LIN {X 0,Y 531.039,Z 315.337,A -85,B 0,C 180,E1 -4242.225,E2 -4242.225} C_VEL
LIN {X 0,Y 530.994,Z 315.34,A -85,B 0,C 180,E1 -4245.35,E2 -4245.35} C_VEL
LIN {X 0,Y 530.991,Z 315.339,A -85,B 0,C 180,E1 -4248.521,E2 -4248.521} C_VEL
LIN {X 0,Y 530.998,Z 315.337,A -85,B 0,C 180,E1 -4250.938,E2 -4250.938} C_VEL
LIN {X 0,Y 530.979,Z 315.343,A -85,B 0,C 180,E1 -4254.225,E2 -4254.225} C_VEL
LIN {X 0,Y 531.004,Z 315.337,A -85,B 0,C 180,E1 -4256.744,E2 -4256.744} C_VEL
LIN {X 0,Y 530.981,Z 315.343,A -85,B 0,C 180,E1 -4259.323,E2 -4259.323} C_VEL
LIN {X 0,Y 530.97,Z 315.344,A -85,B 0,C 180,E1 -4262.102,E2 -4262.102} C_VEL
LIN {X 0,Y 530.986,Z 315.339,A -85,B 0,C 180,E1 -4264.854,E2 -4264.854} C_VEL
LIN {X 0,Y 530.966,Z 315.347,A -85,B 0,C 180,E1 -4267.508,E2 -4267.508} C_VEL
LIN {X 0,Y 530.982,Z 315.34,A -85,B 0,C 180,E1 -4270.433,E2 -4270.433} C_VEL
LIN {X 0,Y 530.961,Z 315.347,A -85,B 0,C 180,E1 -4273.282,E2 -4273.282} C_VEL
LIN {X 0,Y 530.982,Z 315.347,A -85,B 0,C 180,E1 -4275.622,E2 -4275.622} C_VEL
LIN {X 0,Y 530.994,Z 315.338,A -85,B 0,C 180,E1 -4278.565,E2 -4278.565} C_VEL
LIN {X 0,Y 530.958,Z 315.35,A -85,B 0,C 180,E1 -4281.53,E2 -4281.53} C_VEL
LIN {X 0,Y 530.955,Z 315.343,A -85,B 0,C 180,E1 -4284.381,E2 -4284.381} C_VEL
LIN {X 0,Y 530.968,Z 315.345,A -85,B 0,C 180,E1 -4287.134,E2 -4287.134} C_VEL
LIN {X 0,Y 530.964,Z 315.346,A -85,B 0,C 180,E1 -4289.803,E2 -4289.803} C_VEL
LIN {X 0,Y 531.013,Z 315.335,A -85,B 0,C 180,E1 -4292.469,E2 -4292.469} C_VEL
LIN {X 0,Y 531.002,Z 315.339,A -85,B 0,C 180,E1 -4294.943,E2 -4294.943} C_VEL
LIN {X 0,Y 530.969,Z 315.349,A -85,B 0,C 180,E1 -4297.377,E2 -4297.377} C_VEL
LIN {X 0,Y 532.621,Z 320.667,A -85,B 0,C 180,E1 -4297.507,E2 -4297.507} C_VEL
LIN {X 0,Y 532.362,Z 402.902,A -85,B 0,C 180,E1 -4298.663,E2 -4298.663} C_VEL
LIN {X 0,Y 532.209,Z 415.998,A -85,B 0,C 180,E1 -4298.986,E2 -4298.986} C_VEL
LIN {X 0,Y 532.03,Z 429.878,A -85,B 0,C 180,E1 -4299.517,E2 -4299.517} C_VEL
LIN {X 0,Y 531.847,Z 441.157,A -85,B 0,C 180,E1 -4300.107,E2 -4300.107} C_VEL
LIN {X 0,Y 531.61,Z 451.611,A -85,B 0,C 180,E1 -4300.801,E2 -4300.801} C_VEL
LIN {X 0,Y 531.404,Z 461.288,A -85,B 0,C 180,E1 -4301.594,E2 -4301.594} C_VEL
LIN {X 0,Y 531.176,Z 470.826,A -85,B 0,C 180,E1 -4302.552,E2 -4302.552} C_VEL
LIN {X 0,Y 530.961,Z 479.751,A -85,B 0,C 180,E1 -4303.664,E2 -4303.664} C_VEL
LIN {X 0,Y 530.809,Z 487.195,A -85,B 0,C 180,E1 -4304.83,E2 -4304.83} C_VEL
LIN {X 0,Y 530.705,Z 492.339,A -85,B 0,C 180,E1 -4305.819,E2 -4305.819} C_VEL
LIN {X 0,Y 530.574,Z 497.221,A -85,B 0,C 180,E1 -4306.987,E2 -4306.987} C_VEL
LIN {X 0,Y 530.558,Z 500.943,A -85,B 0,C 180,E1 -4308.152,E2 -4308.152} C_VEL
LIN {X 0,Y 530.478,Z 503.626,A -85,B 0,C 180,E1 -4309.311,E2 -4309.311} C_VEL
LIN {X 0,Y 530.462,Z 504.893,A -85,B 0,C 180,E1 -4310.083,E2 -4310.083} C_VEL
LIN {X 0,Y 530.464,Z 505.756,A -85,B 0,C 180,E1 -4310.852,E2 -4310.852} C_VEL
LIN {X 0,Y 530.493,Z 506.174,A -85,B 0,C 180,E1 -4312.387,E2 -4312.387} C_VEL
LIN {X 0,Y 530.548,Z 505.548,A -85,B 0,C 180,E1 -4313.468,E2 -4313.468} C_VEL
LIN {X 0,Y 530.506,Z 503.888,A -85,B 0,C 180,E1 -4314.679,E2 -4314.679} C_VEL
LIN {X 0,Y 530.559,Z 501.365,A -85,B 0,C 180,E1 -4315.822,E2 -4315.822} C_VEL
LIN {X 0,Y 530.61,Z 497.858,A -85,B 0,C 180,E1 -4316.963,E2 -4316.963} C_VEL
LIN {X 0,Y 530.664,Z 493.275,A -85,B 0,C 180,E1 -4318.103,E2 -4318.103} C_VEL
LIN {X 0,Y 530.832,Z 487.475,A -85,B 0,C 180,E1 -4319.242,E2 -4319.242} C_VEL
LIN {X 0,Y 530.951,Z 480.294,A -85,B 0,C 180,E1 -4320.38,E2 -4320.38} C_VEL
LIN {X 0,Y 531.189,Z 471.278,A -85,B 0,C 180,E1 -4321.517,E2 -4321.517} C_VEL
LIN {X 0,Y 531.409,Z 461.946,A -85,B 0,C 180,E1 -4322.464,E2 -4322.464} C_VEL
LIN {X 0,Y 531.655,Z 452.816,A -85,B 0,C 180,E1 -4323.221,E2 -4323.221} C_VEL
LIN {X 0,Y 531.875,Z 443.079,A -85,B 0,C 180,E1 -4323.883,E2 -4323.883} C_VEL
LIN {X 0,Y 532.06,Z 431.73,A -85,B 0,C 180,E1 -4324.499,E2 -4324.499} C_VEL
LIN {X 0,Y 532.19,Z 418.807,A -85,B 0,C 180,E1 -4325.019,E2 -4325.019} C_VEL
LIN {X 0,Y 532.304,Z 405.636,A -85,B 0,C 180,E1 -4325.374,E2 -4325.374} C_VEL
LIN {X 0,Y 532.466,Z 376.911,A -85,B 0,C 180,E1 -4325.8,E2 -4325.8} C_VEL
LIN {X 0,Y 532.689,Z 320.761,A -85,B 0,C 180,E1 -4326.582,E2 -4326.582} C_VEL
LIN {X 0,Y 531.014,Z 315.344,A -85,B 0,C 180,E1 -4326.714,E2 -4326.714} C_VEL
LIN {X 0,Y 530.993,Z 315.343,A -85,B 0,C 180,E1 -4329.139,E2 -4329.139} C_VEL
LIN {X 0,Y 530.972,Z 315.347,A -85,B 0,C 180,E1 -4332.227,E2 -4332.227} C_VEL
LIN {X 0,Y 530.987,Z 315.34,A -85,B 0,C 180,E1 -4335.35,E2 -4335.35} C_VEL
LIN {X 0,Y 530.95,Z 315.351,A -85,B 0,C 180,E1 -4338.523,E2 -4338.523} C_VEL
LIN {X 0,Y 530.931,Z 315.349,A -85,B 0,C 180,E1 -4340.941,E2 -4340.941} C_VEL
LIN {X 0,Y 530.947,Z 315.344,A -85,B 0,C 180,E1 -4343.397,E2 -4343.397} C_VEL
LIN {X 0,Y 530.93,Z 315.351,A -85,B 0,C 180,E1 -4345.902,E2 -4345.902} C_VEL
LIN {X 0,Y 530.933,Z 315.351,A -85,B 0,C 180,E1 -4348.46,E2 -4348.46} C_VEL
LIN {X 0,Y 530.944,Z 315.344,A -85,B 0,C 180,E1 -4351.08,E2 -4351.08} C_VEL
LIN {X 0,Y 530.955,Z 315.347,A -85,B 0,C 180,E1 -4353.775,E2 -4353.775} C_VEL
LIN {X 0,Y 530.911,Z 315.349,A -85,B 0,C 180,E1 -4356.562,E2 -4356.562} C_VEL
LIN {X 0,Y 530.972,Z 315.342,A -85,B 0,C 180,E1 -4359.445,E2 -4359.445} C_VEL
LIN {X 0,Y 530.922,Z 315.348,A -85,B 0,C 180,E1 -4362.463,E2 -4362.463} C_VEL
LIN {X 0,Y 530.97,Z 315.344,A -85,B 0,C 180,E1 -4365.451,E2 -4365.451} C_VEL
LIN {X 0,Y 530.967,Z 315.341,A -85,B 0,C 180,E1 -4368.561,E2 -4368.561} C_VEL
LIN {X 0,Y 530.956,Z 315.349,A -85,B 0,C 180,E1 -4371.529,E2 -4371.529} C_VEL
LIN {X 0,Y 530.952,Z 315.344,A -85,B 0,C 180,E1 -4374.379,E2 -4374.379} C_VEL
LIN {X 0,Y 530.971,Z 315.344,A -85,B 0,C 180,E1 -4377.133,E2 -4377.133} C_VEL
LIN {X 0,Y 530.973,Z 315.347,A -85,B 0,C 180,E1 -4379.803,E2 -4379.803} C_VEL
LIN {X 0,Y 531.024,Z 315.545,A -85,B 0,C 180,E1 -4382.212,E2 -4382.212} C_VEL
LIN {X 0,Y 533.268,Z 326.124,A -85,B 0,C 180,E1 -4383.661,E2 -4383.661} C_VEL
LIN {X 0,Y 532.877,Z 345.545,A -85,B 0,C 180,E1 -4386.074,E2 -4386.074} C_VEL
LIN {X 0,Y 532.428,Z 368.596,A -85,B 0,C 180,E1 -4388.918,E2 -4388.918} C_VEL
LIN {X 0,Y 531.903,Z 396.768,A -85,B 0,C 180,E1 -4392.308,E2 -4392.308} C_VEL
LIN {X 0,Y 531.523,Z 420.074,A -85,B 0,C 180,E1 -4395.053,E2 -4395.053} C_VEL
LIN {X 0,Y 532.776,Z 431.286,A -85,B 0,C 180,E1 -4395.246,E2 -4395.246} C_VEL
LIN {X 0,Y 532.352,Z 528.112,A -85,B 0,C 180,E1 -4396.569,E2 -4396.569} C_VEL
LIN {X 0,Y 532.201,Z 540.608,A -85,B 0,C 180,E1 -4396.857,E2 -4396.857} C_VEL
LIN {X 0,Y 531.959,Z 553.505,A -85,B 0,C 180,E1 -4397.312,E2 -4397.312} C_VEL
LIN {X 0,Y 531.724,Z 565.811,A -85,B 0,C 180,E1 -4397.905,E2 -4397.905} C_VEL
LIN {X 0,Y 531.503,Z 577.756,A -85,B 0,C 180,E1 -4398.656,E2 -4398.656} C_VEL
LIN {X 0,Y 531.256,Z 588.623,A -85,B 0,C 180,E1 -4399.519,E2 -4399.519} C_VEL
LIN {X 0,Y 531.033,Z 598.418,A -85,B 0,C 180,E1 -4400.477,E2 -4400.477} C_VEL
LIN {X 0,Y 530.851,Z 606.454,A -85,B 0,C 180,E1 -4401.434,E2 -4401.434} C_VEL
LIN {X 0,Y 530.682,Z 614.305,A -85,B 0,C 180,E1 -4402.581,E2 -4402.581} C_VEL
LIN {X 0,Y 530.585,Z 621.541,A -85,B 0,C 180,E1 -4403.917,E2 -4403.917} C_VEL
LIN {X 0,Y 530.459,Z 626.318,A -85,B 0,C 180,E1 -4405.06,E2 -4405.06} C_VEL
LIN {X 0,Y 530.516,Z 629.946,A -85,B 0,C 180,E1 -4406.202,E2 -4406.202} C_VEL
LIN {X 0,Y 530.457,Z 631.803,A -85,B 0,C 180,E1 -4406.962,E2 -4406.962} C_VEL
LIN {X 0,Y 530.411,Z 633.192,A -85,B 0,C 180,E1 -4407.722,E2 -4407.722} C_VEL
LIN {X 0,Y 530.344,Z 634.785,A -85,B 0,C 180,E1 -4409.241,E2 -4409.241} C_VEL
LIN {X 0,Y 530.342,Z 635,A -85,B 0,C 180,E1 -4410,E2 -4410} C_VEL
LIN {X 0,Y 530.361,Z 634.183,A -85,B 0,C 180,E1 -4411.519,E2 -4411.519} C_VEL
LIN {X 0,Y 530.411,Z 633.195,A -85,B 0,C 180,E1 -4412.278,E2 -4412.278} C_VEL
LIN {X 0,Y 530.457,Z 631.807,A -85,B 0,C 180,E1 -4413.038,E2 -4413.038} C_VEL
LIN {X 0,Y 530.522,Z 628.876,A -85,B 0,C 180,E1 -4414.178,E2 -4414.178} C_VEL
LIN {X 0,Y 530.525,Z 624.876,A -85,B 0,C 180,E1 -4415.321,E2 -4415.321} C_VEL
LIN {X 0,Y 530.596,Z 619.076,A -85,B 0,C 180,E1 -4416.579,E2 -4416.579} C_VEL
LIN {X 0,Y 530.728,Z 611.833,A -85,B 0,C 180,E1 -4417.801,E2 -4417.801} C_VEL
LIN {X 0,Y 530.908,Z 603.357,A -85,B 0,C 180,E1 -4418.948,E2 -4418.948} C_VEL
LIN {X 0,Y 531.103,Z 594.649,A -85,B 0,C 180,E1 -4419.906,E2 -4419.906} C_VEL
LIN {X 0,Y 531.345,Z 583.897,A -85,B 0,C 180,E1 -4420.864,E2 -4420.864} C_VEL
LIN {X 0,Y 531.559,Z 572.848,A -85,B 0,C 180,E1 -4421.659,E2 -4421.659} C_VEL
LIN {X 0,Y 531.831,Z 561.541,A -85,B 0,C 180,E1 -4422.303,E2 -4422.303} C_VEL
LIN {X 0,Y 532.054,Z 549.413,A -85,B 0,C 180,E1 -4422.831,E2 -4422.831} C_VEL
LIN {X 0,Y 532.213,Z 536.317,A -85,B 0,C 180,E1 -4423.24,E2 -4423.24} C_VEL
LIN {X 0,Y 532.363,Z 524.159,A -85,B 0,C 180,E1 -4423.479,E2 -4423.479} C_VEL
LIN {X 0,Y 532.625,Z 428.755,A -85,B 0,C 180,E1 -4424.776,E2 -4424.776} C_VEL
LIN {X 0,Y 531.483,Z 418.906,A -85,B 0,C 180,E1 -4424.969,E2 -4424.969} C_VEL
LIN {X 0,Y 531.936,Z 388.838,A -85,B 0,C 180,E1 -4428.487,E2 -4428.487} C_VEL
LIN {X 0,Y 532.271,Z 363.451,A -85,B 0,C 180,E1 -4431.494,E2 -4431.494} C_VEL
LIN {X 0,Y 532.637,Z 339.943,A -85,B 0,C 180,E1 -4434.325,E2 -4434.325} C_VEL
LIN {X 0,Y 532.749,Z 324.506,A -85,B 0,C 180,E1 -4436.226,E2 -4436.226} C_VEL
LIN {X 0,Y 530.968,Z 315.346,A -85,B 0,C 180,E1 -4437.466,E2 -4437.466} C_VEL
LIN {X 0,Y 530.972,Z 315.349,A -85,B 0,C 180,E1 -4440.197,E2 -4440.197} C_VEL
LIN {X 0,Y 530.969,Z 315.346,A -85,B 0,C 180,E1 -4442.867,E2 -4442.867} C_VEL
LIN {X 0,Y 530.953,Z 315.345,A -85,B 0,C 180,E1 -4445.62,E2 -4445.62} C_VEL
LIN {X 0,Y 530.966,Z 315.347,A -85,B 0,C 180,E1 -4448.653,E2 -4448.653} C_VEL
LIN {X 0,Y 530.966,Z 315.343,A -85,B 0,C 180,E1 -4451.438,E2 -4451.438} C_VEL
LIN {X 0,Y 530.968,Z 315.345,A -85,B 0,C 180,E1 -4454.549,E2 -4454.549} C_VEL
LIN {X 0,Y 530.932,Z 315.348,A -85,B 0,C 180,E1 -4457.538,E2 -4457.538} C_VEL
LIN {X 0,Y 530.97,Z 315.343,A -85,B 0,C 180,E1 -4460.555,E2 -4460.555} C_VEL
LIN {X 0,Y 530.909,Z 315.35,A -85,B 0,C 180,E1 -4463.437,E2 -4463.437} C_VEL
LIN {X 0,Y 530.953,Z 315.347,A -85,B 0,C 180,E1 -4466.224,E2 -4466.224} C_VEL
LIN {X 0,Y 530.942,Z 315.345,A -85,B 0,C 180,E1 -4468.919,E2 -4468.919} C_VEL
LIN {X 0,Y 530.931,Z 315.352,A -85,B 0,C 180,E1 -4471.54,E2 -4471.54} C_VEL
LIN {X 0,Y 530.93,Z 315.35,A -85,B 0,C 180,E1 -4474.175,E2 -4474.175} C_VEL
LIN {X 0,Y 530.945,Z 315.345,A -85,B 0,C 180,E1 -4476.602,E2 -4476.602} C_VEL
LIN {X 0,Y 530.936,Z 315.349,A -85,B 0,C 180,E1 -4479.059,E2 -4479.059} C_VEL
LIN {X 0,Y 530.956,Z 315.35,A -85,B 0,C 180,E1 -4481.477,E2 -4481.477} C_VEL
LIN {X 0,Y 530.985,Z 315.342,A -85,B 0,C 180,E1 -4484.65,E2 -4484.65} C_VEL
LIN {X 0,Y 530.999,Z 315.346,A -85,B 0,C 180,E1 -4487.361,E2 -4487.361} C_VEL
LIN {X 0,Y 532.788,Z 321.335,A -85,B 0,C 180,E1 -4487.518,E2 -4487.518} C_VEL
LIN {X 0,Y 532.294,Z 404.517,A -85,B 0,C 180,E1 -4488.697,E2 -4488.697} C_VEL
LIN {X 0,Y 532.203,Z 417.459,A -85,B 0,C 180,E1 -4489.033,E2 -4489.033} C_VEL
LIN {X 0,Y 532.055,Z 430.472,A -85,B 0,C 180,E1 -4489.535,E2 -4489.535} C_VEL
LIN {X 0,Y 531.887,Z 441.409,A -85,B 0,C 180,E1 -4490.109,E2 -4490.109} C_VEL
LIN {X 0,Y 531.663,Z 451.53,A -85,B 0,C 180,E1 -4490.777,E2 -4490.777} C_VEL
LIN {X 0,Y 531.479,Z 460.939,A -85,B 0,C 180,E1 -4491.54,E2 -4491.54} C_VEL
LIN {X 0,Y 531.243,Z 469.664,A -85,B 0,C 180,E1 -4492.398,E2 -4492.398} C_VEL
LIN {X 0,Y 531.087,Z 477.845,A -85,B 0,C 180,E1 -4493.377,E2 -4493.377} C_VEL
LIN {X 0,Y 530.922,Z 485.456,A -85,B 0,C 180,E1 -4494.492,E2 -4494.492} C_VEL
LIN {X 0,Y 530.765,Z 490.739,A -85,B 0,C 180,E1 -4495.443,E2 -4495.443} C_VEL
LIN {X 0,Y 530.69,Z 495.884,A -85,B 0,C 180,E1 -4496.583,E2 -4496.583} C_VEL
LIN {X 0,Y 530.513,Z 499.891,A -85,B 0,C 180,E1 -4497.722,E2 -4497.722} C_VEL
LIN {X 0,Y 530.49,Z 501.978,A -85,B 0,C 180,E1 -4498.481,E2 -4498.481} C_VEL
LIN {X 0,Y 530.434,Z 504.873,A -85,B 0,C 180,E1 -4500,E2 -4500} C_VEL
LIN {X 0,Y 530.435,Z 505.724,A -85,B 0,C 180,E1 -4500.759,E2 -4500.759} C_VEL
LIN {X 0,Y 530.443,Z 506.227,A -85,B 0,C 180,E1 -4502.278,E2 -4502.278} C_VEL
LIN {X 0,Y 530.527,Z 505.908,A -85,B 0,C 180,E1 -4503.037,E2 -4503.037} C_VEL
LIN {X 0,Y 530.495,Z 504.062,A -85,B 0,C 180,E1 -4504.559,E2 -4504.559} C_VEL
LIN {X 0,Y 530.551,Z 501.611,A -85,B 0,C 180,E1 -4505.701,E2 -4505.701} C_VEL
LIN {X 0,Y 530.636,Z 498.166,A -85,B 0,C 180,E1 -4506.846,E2 -4506.846} C_VEL
LIN {X 0,Y 530.677,Z 493.63,A -85,B 0,C 180,E1 -4507.993,E2 -4507.993} C_VEL
LIN {X 0,Y 530.816,Z 487.858,A -85,B 0,C 180,E1 -4509.142,E2 -4509.142} C_VEL
LIN {X 0,Y 530.976,Z 480.662,A -85,B 0,C 180,E1 -4510.293,E2 -4510.293} C_VEL
LIN {X 0,Y 531.142,Z 471.64,A -85,B 0,C 180,E1 -4511.448,E2 -4511.448} C_VEL
LIN {X 0,Y 531.35,Z 462.198,A -85,B 0,C 180,E1 -4512.411,E2 -4512.411} C_VEL
LIN {X 0,Y 531.568,Z 452.971,A -85,B 0,C 180,E1 -4513.183,E2 -4513.183} C_VEL
LIN {X 0,Y 531.782,Z 443.105,A -85,B 0,C 180,E1 -4513.859,E2 -4513.859} C_VEL
LIN {X 0,Y 532.005,Z 432.573,A -85,B 0,C 180,E1 -4514.438,E2 -4514.438} C_VEL
LIN {X 0,Y 532.195,Z 421.184,A -85,B 0,C 180,E1 -4514.922,E2 -4514.922} C_VEL
LIN {X 0,Y 532.291,Z 408.39,A -85,B 0,C 180,E1 -4515.311,E2 -4515.311} C_VEL
LIN {X 0,Y 532.389,Z 394.101,A -85,B 0,C 180,E1 -4515.564,E2 -4515.564} C_VEL
LIN {X 0,Y 532.621,Z 320.586,A -85,B 0,C 180,E1 -4516.585,E2 -4516.585} C_VEL
LIN {X 0,Y 530.987,Z 315.347,A -85,B 0,C 180,E1 -4516.706,E2 -4516.706} C_VEL
LIN {X 0,Y 531.034,Z 315.334,A -85,B 0,C 180,E1 -4520.006,E2 -4520.006} C_VEL
LIN {X 0,Y 530.946,Z 315.351,A -85,B 0,C 180,E1 -4522.573,E2 -4522.573} C_VEL
LIN {X 0,Y 531.005,Z 315.339,A -85,B 0,C 180,E1 -4525.057,E2 -4525.057} C_VEL
LIN {X 0,Y 531.014,Z 315.335,A -85,B 0,C 180,E1 -4527.595,E2 -4527.595} C_VEL
LIN {X 0,Y 530.967,Z 315.35,A -85,B 0,C 180,E1 -4530.643,E2 -4530.643} C_VEL
LIN {X 0,Y 530.952,Z 315.343,A -85,B 0,C 180,E1 -4531.757,E2 -4531.757} C_VEL
LIN {X 0,Y 530.318,Z 315.429,A -85,B 0,C 180,E1 -4532.39,E2 -4532.39} C_VEL
LIN {X 0,Y 527.482,Z 315.782,A -85,B 0,C 180,E1 -4533.419,E2 -4533.419} C_VEL
LIN {X 0,Y 525.062,Z 316.083,A -85,B 0,C 180,E1 -4534.247,E2 -4534.247} C_VEL
LIN {X 0,Y 524.012,Z 316.212,A -85,B 0,C 180,E1 -4534.886,E2 -4534.886} C_VEL
LIN {X 0,Y 523.923,Z 316.22,A -85,B 0,C 180,E1 -4535.102,E2 -4535.102} C_VEL
LIN {X 0,Y 523.915,Z 316.223,A -85,B 0,C 180,E1 -4538.101,E2 -4538.101} C_VEL
LIN {X 0,Y 523.938,Z 316.218,A -85,B 0,C 180,E1 -4541.092,E2 -4541.092} C_VEL
LIN {X 0,Y 523.935,Z 316.222,A -85,B 0,C 180,E1 -4544.228,E2 -4544.228} C_VEL
LIN {X 0,Y 523.915,Z 316.223,A -85,B 0,C 180,E1 -4546.832,E2 -4546.832} C_VEL
LIN {X 0,Y 523.937,Z 316.219,A -85,B 0,C 180,E1 -4548.907,E2 -4548.907} C_VEL
LIN {X 0,Y 523.915,Z 316.222,A -85,B 0,C 180,E1 -4551.898,E2 -4551.898} C_VEL
LIN {X 0,Y 523.935,Z 316.219,A -85,B 0,C 180,E1 -4554.909,E2 -4554.909} C_VEL
LIN {X 0,Y 523.936,Z 316.218,A -85,B 0,C 180,E1 -4557.679,E2 -4557.679} C_VEL
LIN {X 0,Y 523.952,Z 316.219,A -85,B 0,C 180,E1 -4560.676,E2 -4560.676} C_VEL
LIN {X 0,Y 523.973,Z 316.214,A -85,B 0,C 180,E1 -4563.728,E2 -4563.728} C_VEL
LIN {X 0,Y 523.935,Z 316.225,A -85,B 0,C 180,E1 -4566.271,E2 -4566.271} C_VEL
LIN {X 0,Y 523.944,Z 316.218,A -85,B 0,C 180,E1 -4568.767,E2 -4568.767} C_VEL
LIN {X 0,Y 523.951,Z 316.215,A -85,B 0,C 180,E1 -4571.221,E2 -4571.221} C_VEL
LIN {X 0,Y 523.934,Z 316.219,A -85,B 0,C 180,E1 -4573.639,E2 -4573.639} C_VEL
LIN {X 0,Y 523.938,Z 316.223,A -85,B 0,C 180,E1 -4576.028,E2 -4576.028} C_VEL
LIN {X 0,Y 524.01,Z 316.213,A -85,B 0,C 180,E1 -4578.394,E2 -4578.394} C_VEL
LIN {X 0,Y 524.001,Z 316.21,A -85,B 0,C 180,E1 -4581.516,E2 -4581.516} C_VEL
LIN {X 0,Y 524.08,Z 316.201,A -85,B 0,C 180,E1 -4584.614,E2 -4584.614} C_VEL
LIN {X 0,Y 524.111,Z 316.199,A -85,B 0,C 180,E1 -4587.695,E2 -4587.695} C_VEL
LIN {X 0,Y 524.121,Z 316.194,A -85,B 0,C 180,E1 -4590.768,E2 -4590.768} C_VEL
LIN {X 0,Y 524.069,Z 316.2,A -85,B 0,C 180,E1 -4593.075,E2 -4593.075} C_VEL
LIN {X 0,Y 524.044,Z 316.21,A -85,B 0,C 180,E1 -4596.159,E2 -4596.159} C_VEL
LIN {X 0,Y 523.996,Z 316.211,A -85,B 0,C 180,E1 -4599.262,E2 -4599.262} C_VEL
LIN {X 0,Y 524.001,Z 316.215,A -85,B 0,C 180,E1 -4601.74,E2 -4601.74} C_VEL
LIN {X 0,Y 523.991,Z 316.21,A -85,B 0,C 180,E1 -4605.053,E2 -4605.053} C_VEL
LIN {X 0,Y 523.963,Z 316.221,A -85,B 0,C 180,E1 -4607.969,E2 -4607.969} C_VEL
LIN {X 0,Y 523.97,Z 316.214,A -85,B 0,C 180,E1 -4610.41,E2 -4610.41} C_VEL
LIN {X 0,Y 523.916,Z 316.22,A -85,B 0,C 180,E1 -4612.894,E2 -4612.894} C_VEL
LIN {X 0,Y 523.952,Z 316.219,A -85,B 0,C 180,E1 -4615.419,E2 -4615.419} C_VEL
LIN {X 0,Y 523.968,Z 316.218,A -85,B 0,C 180,E1 -4617.999,E2 -4617.999} C_VEL
LIN {X 0,Y 523.944,Z 316.216,A -85,B 0,C 180,E1 -4620.855,E2 -4620.855} C_VEL
LIN {X 0,Y 523.961,Z 316.222,A -85,B 0,C 180,E1 -4623.735,E2 -4623.735} C_VEL
LIN {X 0,Y 523.919,Z 316.22,A -85,B 0,C 180,E1 -4626.404,E2 -4626.404} C_VEL
LIN {X 0,Y 523.922,Z 316.221,A -85,B 0,C 180,E1 -4629.085,E2 -4629.085} C_VEL
LIN {X 0,Y 523.951,Z 316.218,A -85,B 0,C 180,E1 -4632.12,E2 -4632.12} C_VEL
LIN {X 0,Y 523.946,Z 316.221,A -85,B 0,C 180,E1 -4635.31,E2 -4635.31} C_VEL
LIN {X 0,Y 523.956,Z 316.215,A -85,B 0,C 180,E1 -4638.69,E2 -4638.69} C_VEL
LIN {X 0,Y 523.918,Z 316.222,A -85,B 0,C 180,E1 -4641.081,E2 -4641.081} C_VEL
LIN {X 0,Y 523.902,Z 316.226,A -85,B 0,C 180,E1 -4643.826,E2 -4643.826} C_VEL
LIN {X 0,Y 523.915,Z 316.22,A -85,B 0,C 180,E1 -4646.634,E2 -4646.634} C_VEL
LIN {X 0,Y 523.951,Z 316.221,A -85,B 0,C 180,E1 -4649.356,E2 -4649.356} C_VEL
LIN {X 0,Y 523.978,Z 316.212,A -85,B 0,C 180,E1 -4652.283,E2 -4652.283} C_VEL
LIN {X 0,Y 523.951,Z 316.215,A -85,B 0,C 180,E1 -4654.582,E2 -4654.582} C_VEL
LIN {X 0,Y 523.948,Z 316.223,A -85,B 0,C 180,E1 -4657.18,E2 -4657.18} C_VEL
LIN {X 0,Y 525.86,Z 323.012,A -85,B 0,C 180,E1 -4657.347,E2 -4657.347} C_VEL
LIN {X 0,Y 525.472,Z 403.568,A -85,B 0,C 180,E1 -4658.498,E2 -4658.498} C_VEL
LIN {X 0,Y 525.297,Z 416.648,A -85,B 0,C 180,E1 -4658.824,E2 -4658.824} C_VEL
LIN {X 0,Y 525.154,Z 429.634,A -85,B 0,C 180,E1 -4659.321,E2 -4659.321} C_VEL
LIN {X 0,Y 524.94,Z 441.47,A -85,B 0,C 180,E1 -4659.936,E2 -4659.936} C_VEL
LIN {X 0,Y 524.676,Z 452.036,A -85,B 0,C 180,E1 -4660.639,E2 -4660.639} C_VEL
LIN {X 0,Y 524.466,Z 461.781,A -85,B 0,C 180,E1 -4661.443,E2 -4661.443} C_VEL
LIN {X 0,Y 524.229,Z 471.143,A -85,B 0,C 180,E1 -4662.388,E2 -4662.388} C_VEL
LIN {X 0,Y 523.992,Z 479.646,A -85,B 0,C 180,E1 -4663.441,E2 -4663.441} C_VEL
LIN {X 0,Y 523.82,Z 487.444,A -85,B 0,C 180,E1 -4664.646,E2 -4664.646} C_VEL
LIN {X 0,Y 523.708,Z 492.611,A -85,B 0,C 180,E1 -4665.626,E2 -4665.626} C_VEL
LIN {X 0,Y 523.555,Z 497.621,A -85,B 0,C 180,E1 -4666.809,E2 -4666.809} C_VEL
LIN {X 0,Y 523.546,Z 501.458,A -85,B 0,C 180,E1 -4667.991,E2 -4667.991} C_VEL
LIN {X 0,Y 523.464,Z 504.248,A -85,B 0,C 180,E1 -4669.166,E2 -4669.166} C_VEL
LIN {X 0,Y 523.418,Z 505.594,A -85,B 0,C 180,E1 -4669.948,E2 -4669.948} C_VEL
LIN {X 0,Y 523.435,Z 506.485,A -85,B 0,C 180,E1 -4670.728,E2 -4670.728} C_VEL
LIN {X 0,Y 523.458,Z 507.059,A -85,B 0,C 180,E1 -4672.284,E2 -4672.284} C_VEL
LIN {X 0,Y 523.505,Z 506.452,A -85,B 0,C 180,E1 -4673.439,E2 -4673.439} C_VEL
LIN {X 0,Y 523.486,Z 504.941,A -85,B 0,C 180,E1 -4674.608,E2 -4674.608} C_VEL
LIN {X 0,Y 523.523,Z 503.431,A -85,B 0,C 180,E1 -4675.38,E2 -4675.38} C_VEL
LIN {X 0,Y 523.596,Z 500.353,A -85,B 0,C 180,E1 -4676.538,E2 -4676.538} C_VEL
LIN {X 0,Y 523.622,Z 496.249,A -85,B 0,C 180,E1 -4677.693,E2 -4677.693} C_VEL
LIN {X 0,Y 523.756,Z 489.962,A -85,B 0,C 180,E1 -4679.039,E2 -4679.039} C_VEL
LIN {X 0,Y 523.952,Z 483.092,A -85,B 0,C 180,E1 -4680.192,E2 -4680.192} C_VEL
LIN {X 0,Y 524.168,Z 474.577,A -85,B 0,C 180,E1 -4681.345,E2 -4681.345} C_VEL
LIN {X 0,Y 524.45,Z 464.799,A -85,B 0,C 180,E1 -4682.4,E2 -4682.4} C_VEL
LIN {X 0,Y 524.718,Z 453.656,A -85,B 0,C 180,E1 -4683.36,E2 -4683.36} C_VEL
LIN {X 0,Y 524.953,Z 443.896,A -85,B 0,C 180,E1 -4684.031,E2 -4684.031} C_VEL
LIN {X 0,Y 525.142,Z 432.447,A -85,B 0,C 180,E1 -4684.654,E2 -4684.654} C_VEL
LIN {X 0,Y 525.285,Z 419.445,A -85,B 0,C 180,E1 -4685.182,E2 -4685.182} C_VEL
LIN {X 0,Y 525.374,Z 407.352,A -85,B 0,C 180,E1 -4685.518,E2 -4685.518} C_VEL
LIN {X 0,Y 525.543,Z 382.309,A -85,B 0,C 180,E1 -4685.901,E2 -4685.901} C_VEL
LIN {X 0,Y 525.776,Z 321.915,A -85,B 0,C 180,E1 -4686.763,E2 -4686.763} C_VEL
LIN {X 0,Y 523.979,Z 316.219,A -85,B 0,C 180,E1 -4686.909,E2 -4686.909} C_VEL
LIN {X 0,Y 523.945,Z 316.221,A -85,B 0,C 180,E1 -4689.263,E2 -4689.263} C_VEL
LIN {X 0,Y 523.925,Z 316.227,A -85,B 0,C 180,E1 -4692.394,E2 -4692.394} C_VEL
LIN {X 0,Y 523.919,Z 316.221,A -85,B 0,C 180,E1 -4695.563,E2 -4695.563} C_VEL
LIN {X 0,Y 523.912,Z 316.225,A -85,B 0,C 180,E1 -4697.971,E2 -4697.971} C_VEL
LIN {X 0,Y 523.906,Z 316.229,A -85,B 0,C 180,E1 -4700.413,E2 -4700.413} C_VEL
LIN {X 0,Y 523.902,Z 316.223,A -85,B 0,C 180,E1 -4702.894,E2 -4702.894} C_VEL
LIN {X 0,Y 523.881,Z 316.225,A -85,B 0,C 180,E1 -4705.423,E2 -4705.423} C_VEL
LIN {X 0,Y 523.899,Z 316.228,A -85,B 0,C 180,E1 -4708.003,E2 -4708.003} C_VEL
LIN {X 0,Y 523.908,Z 316.222,A -85,B 0,C 180,E1 -4710.847,E2 -4710.847} C_VEL
LIN {X 0,Y 523.931,Z 316.221,A -85,B 0,C 180,E1 -4713.729,E2 -4713.729} C_VEL
LIN {X 0,Y 523.865,Z 316.228,A -85,B 0,C 180,E1 -4716.395,E2 -4716.395} C_VEL
LIN {X 0,Y 523.915,Z 316.218,A -85,B 0,C 180,E1 -4719.086,E2 -4719.086} C_VEL
LIN {X 0,Y 523.902,Z 316.226,A -85,B 0,C 180,E1 -4722.124,E2 -4722.124} C_VEL
LIN {X 0,Y 523.94,Z 316.219,A -85,B 0,C 180,E1 -4725.311,E2 -4725.311} C_VEL
LIN {X 0,Y 523.927,Z 316.218,A -85,B 0,C 180,E1 -4728.694,E2 -4728.694} C_VEL
LIN {X 0,Y 523.915,Z 316.226,A -85,B 0,C 180,E1 -4731.898,E2 -4731.898} C_VEL
LIN {X 0,Y 523.925,Z 316.22,A -85,B 0,C 180,E1 -4734.912,E2 -4734.912} C_VEL
LIN {X 0,Y 523.939,Z 316.224,A -85,B 0,C 180,E1 -4737.68,E2 -4737.68} C_VEL
LIN {X 0,Y 523.957,Z 316.217,A -85,B 0,C 180,E1 -4740.677,E2 -4740.677} C_VEL
LIN {X 0,Y 523.973,Z 316.243,A -85,B 0,C 180,E1 -4741.974,E2 -4741.974} C_VEL
LIN {X 0,Y 526.436,Z 328.106,A -85,B 0,C 180,E1 -4743.624,E2 -4743.624} C_VEL
LIN {X 0,Y 525.923,Z 348.201,A -85,B 0,C 180,E1 -4746.156,E2 -4746.156} C_VEL
LIN {X 0,Y 525.361,Z 372.943,A -85,B 0,C 180,E1 -4749.244,E2 -4749.244} C_VEL
LIN {X 0,Y 524.853,Z 399.403,A -85,B 0,C 180,E1 -4752.465,E2 -4752.465} C_VEL
LIN {X 0,Y 524.446,Z 419.066,A -85,B 0,C 180,E1 -4754.836,E2 -4754.836} C_VEL
LIN {X 0,Y 525.864,Z 432.123,A -85,B 0,C 180,E1 -4755.079,E2 -4755.079} C_VEL
LIN {X 0,Y 525.447,Z 526.339,A -85,B 0,C 180,E1 -4756.389,E2 -4756.389} C_VEL
LIN {X 0,Y 525.25,Z 539.225,A -85,B 0,C 180,E1 -4756.68,E2 -4756.68} C_VEL
LIN {X 0,Y 525.011,Z 552.314,A -85,B 0,C 180,E1 -4757.141,E2 -4757.141} C_VEL
LIN {X 0,Y 524.724,Z 564.892,A -85,B 0,C 180,E1 -4757.752,E2 -4757.752} C_VEL
LIN {X 0,Y 524.48,Z 576.725,A -85,B 0,C 180,E1 -4758.502,E2 -4758.502} C_VEL
LIN {X 0,Y 524.234,Z 587.636,A -85,B 0,C 180,E1 -4759.377,E2 -4759.377} C_VEL
LIN {X 0,Y 523.962,Z 597.46,A -85,B 0,C 180,E1 -4760.348,E2 -4760.348} C_VEL
LIN {X 0,Y 523.771,Z 605.524,A -85,B 0,C 180,E1 -4761.318,E2 -4761.318} C_VEL
LIN {X 0,Y 523.629,Z 613.413,A -85,B 0,C 180,E1 -4762.48,E2 -4762.48} C_VEL
LIN {X 0,Y 523.468,Z 620.046,A -85,B 0,C 180,E1 -4763.706,E2 -4763.706} C_VEL
LIN {X 0,Y 523.461,Z 624.036,A -85,B 0,C 180,E1 -4764.607,E2 -4764.607} C_VEL
LIN {X 0,Y 523.441,Z 628.097,A -85,B 0,C 180,E1 -4765.765,E2 -4765.765} C_VEL
LIN {X 0,Y 523.397,Z 631.091,A -85,B 0,C 180,E1 -4766.921,E2 -4766.921} C_VEL
LIN {X 0,Y 523.338,Z 632.513,A -85,B 0,C 180,E1 -4767.691,E2 -4767.691} C_VEL
LIN {X 0,Y 523.272,Z 634.144,A -85,B 0,C 180,E1 -4769.23,E2 -4769.23} C_VEL
LIN {X 0,Y 523.272,Z 634.361,A -85,B 0,C 180,E1 -4770,E2 -4770} C_VEL
LIN {X 0,Y 523.273,Z 634.138,A -85,B 0,C 180,E1 -4770.769,E2 -4770.769} C_VEL
LIN {X 0,Y 523.339,Z 632.499,A -85,B 0,C 180,E1 -4772.309,E2 -4772.309} C_VEL
LIN {X 0,Y 523.397,Z 631.065,A -85,B 0,C 180,E1 -4773.079,E2 -4773.079} C_VEL
LIN {X 0,Y 523.441,Z 628.051,A -85,B 0,C 180,E1 -4774.235,E2 -4774.235} C_VEL
LIN {X 0,Y 523.461,Z 623.962,A -85,B 0,C 180,E1 -4775.393,E2 -4775.393} C_VEL
LIN {X 0,Y 523.517,Z 618.583,A -85,B 0,C 180,E1 -4776.574,E2 -4776.574} C_VEL
LIN {X 0,Y 523.649,Z 612.064,A -85,B 0,C 180,E1 -4777.713,E2 -4777.713} C_VEL
LIN {X 0,Y 523.821,Z 603.802,A -85,B 0,C 180,E1 -4778.876,E2 -4778.876} C_VEL
LIN {X 0,Y 524.014,Z 595.371,A -85,B 0,C 180,E1 -4779.846,E2 -4779.846} C_VEL
LIN {X 0,Y 524.232,Z 585.055,A -85,B 0,C 180,E1 -4780.818,E2 -4780.818} C_VEL
LIN {X 0,Y 524.487,Z 573.466,A -85,B 0,C 180,E1 -4781.688,E2 -4781.688} C_VEL
LIN {X 0,Y 524.785,Z 561.957,A -85,B 0,C 180,E1 -4782.373,E2 -4782.373} C_VEL
LIN {X 0,Y 525.005,Z 550.374,A -85,B 0,C 180,E1 -4782.908,E2 -4782.908} C_VEL
LIN {X 0,Y 525.216,Z 537.219,A -85,B 0,C 180,E1 -4783.346,E2 -4783.346} C_VEL
LIN {X 0,Y 525.427,Z 523.289,A -85,B 0,C 180,E1 -4783.636,E2 -4783.636} C_VEL
LIN {X 0,Y 525.734,Z 429.558,A -85,B 0,C 180,E1 -4784.944,E2 -4784.944} C_VEL
LIN {X 0,Y 524.413,Z 417.911,A -85,B 0,C 180,E1 -4785.161,E2 -4785.161} C_VEL
LIN {X 0,Y 524.888,Z 389.605,A -85,B 0,C 180,E1 -4788.522,E2 -4788.522} C_VEL
LIN {X 0,Y 525.272,Z 364.094,A -85,B 0,C 180,E1 -4791.589,E2 -4791.589} C_VEL
LIN {X 0,Y 525.662,Z 340.44,A -85,B 0,C 180,E1 -4794.486,E2 -4794.486} C_VEL
LIN {X 0,Y 525.889,Z 327.008,A -85,B 0,C 180,E1 -4796.169,E2 -4796.169} C_VEL
LIN {X 0,Y 524.745,Z 320.158,A -85,B 0,C 180,E1 -4797.089,E2 -4797.089} C_VEL
LIN {X 0,Y 523.927,Z 316.224,A -85,B 0,C 180,E1 -4797.656,E2 -4797.656} C_VEL
LIN {X 0,Y 523.959,Z 316.224,A -85,B 0,C 180,E1 -4800.644,E2 -4800.644} C_VEL
LIN {X 0,Y 523.934,Z 316.221,A -85,B 0,C 180,E1 -4803.73,E2 -4803.73} C_VEL
LIN {X 0,Y 523.902,Z 316.229,A -85,B 0,C 180,E1 -4806.401,E2 -4806.401} C_VEL
LIN {X 0,Y 523.915,Z 316.222,A -85,B 0,C 180,E1 -4809.085,E2 -4809.085} C_VEL
LIN {X 0,Y 523.912,Z 316.228,A -85,B 0,C 180,E1 -4812.123,E2 -4812.123} C_VEL
LIN {X 0,Y 523.938,Z 316.218,A -85,B 0,C 180,E1 -4815.311,E2 -4815.311} C_VEL
LIN {X 0,Y 523.923,Z 316.22,A -85,B 0,C 180,E1 -4818.694,E2 -4818.694} C_VEL
LIN {X 0,Y 523.903,Z 316.228,A -85,B 0,C 180,E1 -4821.897,E2 -4821.897} C_VEL
LIN {X 0,Y 523.916,Z 316.22,A -85,B 0,C 180,E1 -4824.913,E2 -4824.913} C_VEL
LIN {X 0,Y 523.933,Z 316.224,A -85,B 0,C 180,E1 -4827.681,E2 -4827.681} C_VEL
LIN {X 0,Y 523.937,Z 316.218,A -85,B 0,C 180,E1 -4830.68,E2 -4830.68} C_VEL
LIN {X 0,Y 523.883,Z 316.232,A -85,B 0,C 180,E1 -4833.723,E2 -4833.723} C_VEL
LIN {X 0,Y 523.907,Z 316.224,A -85,B 0,C 180,E1 -4836.269,E2 -4836.269} C_VEL
LIN {X 0,Y 523.902,Z 316.223,A -85,B 0,C 180,E1 -4838.764,E2 -4838.764} C_VEL
LIN {X 0,Y 523.915,Z 316.225,A -85,B 0,C 180,E1 -4841.219,E2 -4841.219} C_VEL
LIN {X 0,Y 523.891,Z 316.231,A -85,B 0,C 180,E1 -4843.637,E2 -4843.637} C_VEL
LIN {X 0,Y 523.918,Z 316.225,A -85,B 0,C 180,E1 -4846.027,E2 -4846.027} C_VEL
LIN {X 0,Y 523.957,Z 316.223,A -85,B 0,C 180,E1 -4847.184,E2 -4847.184} C_VEL
LIN {X 0,Y 525.923,Z 322.856,A -85,B 0,C 180,E1 -4847.344,E2 -4847.344} C_VEL
LIN {X 0,Y 525.366,Z 405.685,A -85,B 0,C 180,E1 -4848.546,E2 -4848.546} C_VEL
LIN {X 0,Y 525.277,Z 418.539,A -85,B 0,C 180,E1 -4848.886,E2 -4848.886} C_VEL
LIN {X 0,Y 525.133,Z 431.533,A -85,B 0,C 180,E1 -4849.396,E2 -4849.396} C_VEL
LIN {X 0,Y 524.965,Z 442.465,A -85,B 0,C 180,E1 -4849.977,E2 -4849.977} C_VEL
LIN {X 0,Y 524.691,Z 453.847,A -85,B 0,C 180,E1 -4850.75,E2 -4850.75} C_VEL
LIN {X 0,Y 524.473,Z 464.07,A -85,B 0,C 180,E1 -4851.62,E2 -4851.62} C_VEL
LIN {X 0,Y 524.222,Z 473.009,A -85,B 0,C 180,E1 -4852.556,E2 -4852.556} C_VEL
LIN {X 0,Y 523.986,Z 481.581,A -85,B 0,C 180,E1 -4853.668,E2 -4853.668} C_VEL
LIN {X 0,Y 523.923,Z 488.631,A -85,B 0,C 180,E1 -4854.805,E2 -4854.805} C_VEL
LIN {X 0,Y 523.735,Z 493.527,A -85,B 0,C 180,E1 -4855.767,E2 -4855.767} C_VEL
LIN {X 0,Y 523.586,Z 498.258,A -85,B 0,C 180,E1 -4856.922,E2 -4856.922} C_VEL
LIN {X 0,Y 523.579,Z 501.882,A -85,B 0,C 180,E1 -4858.077,E2 -4858.077} C_VEL
LIN {X 0,Y 523.422,Z 504.532,A -85,B 0,C 180,E1 -4859.23,E2 -4859.23} C_VEL
LIN {X 0,Y 523.407,Z 505.785,A -85,B 0,C 180,E1 -4860,E2 -4860} C_VEL
LIN {X 0,Y 523.411,Z 506.621,A -85,B 0,C 180,E1 -4860.769,E2 -4860.769} C_VEL
LIN {X 0,Y 523.399,Z 507.083,A -85,B 0,C 180,E1 -4862.308,E2 -4862.308} C_VEL
LIN {X 0,Y 523.479,Z 506.741,A -85,B 0,C 180,E1 -4863.078,E2 -4863.078} C_VEL
LIN {X 0,Y 523.464,Z 504.849,A -85,B 0,C 180,E1 -4864.62,E2 -4864.62} C_VEL
LIN {X 0,Y 523.54,Z 502.357,A -85,B 0,C 180,E1 -4865.778,E2 -4865.778} C_VEL
LIN {X 0,Y 523.609,Z 498.87,A -85,B 0,C 180,E1 -4866.938,E2 -4866.938} C_VEL
LIN {X 0,Y 523.659,Z 494.284,A -85,B 0,C 180,E1 -4868.101,E2 -4868.101} C_VEL
LIN {X 0,Y 523.82,Z 488.456,A -85,B 0,C 180,E1 -4869.265,E2 -4869.265} C_VEL
LIN {X 0,Y 524,Z 481.161,A -85,B 0,C 180,E1 -4870.431,E2 -4870.431} C_VEL
LIN {X 0,Y 524.182,Z 472.033,A -85,B 0,C 180,E1 -4871.602,E2 -4871.602} C_VEL
LIN {X 0,Y 524.408,Z 462.486,A -85,B 0,C 180,E1 -4872.578,E2 -4872.578} C_VEL
LIN {X 0,Y 524.677,Z 451.848,A -85,B 0,C 180,E1 -4873.458,E2 -4873.458} C_VEL
LIN {X 0,Y 524.919,Z 441.555,A -85,B 0,C 180,E1 -4874.143,E2 -4874.143} C_VEL
LIN {X 0,Y 525.181,Z 429.301,A -85,B 0,C 180,E1 -4874.779,E2 -4874.779} C_VEL
LIN {X 0,Y 525.355,Z 415.596,A -85,B 0,C 180,E1 -4875.292,E2 -4875.292} C_VEL
LIN {X 0,Y 525.458,Z 403.596,A -85,B 0,C 180,E1 -4875.59,E2 -4875.59} C_VEL
LIN {X 0,Y 525.761,Z 321.988,A -85,B 0,C 180,E1 -4876.759,E2 -4876.759} C_VEL
LIN {X 0,Y 523.959,Z 316.222,A -85,B 0,C 180,E1 -4876.912,E2 -4876.912} C_VEL
LIN {X 0,Y 523.981,Z 316.214,A -85,B 0,C 180,E1 -4880.134,E2 -4880.134} C_VEL
LIN {X 0,Y 523.911,Z 316.225,A -85,B 0,C 180,E1 -4882.893,E2 -4882.893} C_VEL
LIN {X 0,Y 523.953,Z 316.215,A -85,B 0,C 180,E1 -4885.418,E2 -4885.418} C_VEL
LIN {X 0,Y 523.965,Z 316.214,A -85,B 0,C 180,E1 -4887.999,E2 -4887.999} C_VEL
LIN {X 0,Y 523.94,Z 316.221,A -85,B 0,C 180,E1 -4890.853,E2 -4890.853} C_VEL
LIN {X 0,Y 523.93,Z 316.218,A -85,B 0,C 180,E1 -4893.729,E2 -4893.729} C_VEL
LIN {X 0,Y 523.923,Z 316.22,A -85,B 0,C 180,E1 -4895.102,E2 -4895.102} C_VEL
LIN {X 0,Y 523.242,Z 316.304,A -85,B 0,C 180,E1 -4895.743,E2 -4895.743} C_VEL
LIN {X 0,Y 520.374,Z 316.666,A -85,B 0,C 180,E1 -4896.783,E2 -4896.783} C_VEL
LIN {X 0,Y 517.966,Z 316.963,A -85,B 0,C 180,E1 -4897.621,E2 -4897.621} C_VEL
LIN {X 0,Y 516.946,Z 317.092,A -85,B 0,C 180,E1 -4898.268,E2 -4898.268} C_VEL
LIN {X 0,Y 516.87,Z 317.101,A -85,B 0,C 180,E1 -4898.487,E2 -4898.487} C_VEL
LIN {X 0,Y 516.91,Z 317.093,A -85,B 0,C 180,E1 -4901.775,E2 -4901.775} C_VEL
LIN {X 0,Y 516.893,Z 317.096,A -85,B 0,C 180,E1 -4905.007,E2 -4905.007} C_VEL
LIN {X 0,Y 516.912,Z 317.099,A -85,B 0,C 180,E1 -4908.398,E2 -4908.398} C_VEL
LIN {X 0,Y 516.88,Z 317.096,A -85,B 0,C 180,E1 -4911.284,E2 -4911.284} C_VEL
LIN {X 0,Y 516.887,Z 317.101,A -85,B 0,C 180,E1 -4914.221,E2 -4914.221} C_VEL
LIN {X 0,Y 516.895,Z 317.095,A -85,B 0,C 180,E1 -4917.053,E2 -4917.053} C_VEL
LIN {X 0,Y 516.89,Z 317.097,A -85,B 0,C 180,E1 -4919.796,E2 -4919.796} C_VEL
LIN {X 0,Y 516.926,Z 317.097,A -85,B 0,C 180,E1 -4922.467,E2 -4922.467} C_VEL
LIN {X 0,Y 516.909,Z 317.093,A -85,B 0,C 180,E1 -4925.072,E2 -4925.072} C_VEL
LIN {X 0,Y 516.884,Z 317.101,A -85,B 0,C 180,E1 -4928.462,E2 -4928.462} C_VEL
LIN {X 0,Y 516.902,Z 317.094,A -85,B 0,C 180,E1 -4930.955,E2 -4930.955} C_VEL
LIN {X 0,Y 516.911,Z 317.093,A -85,B 0,C 180,E1 -4933.41,E2 -4933.41} C_VEL
LIN {X 0,Y 516.893,Z 317.099,A -85,B 0,C 180,E1 -4935.834,E2 -4935.834} C_VEL
LIN {X 0,Y 516.963,Z 317.093,A -85,B 0,C 180,E1 -4938.234,E2 -4938.234} C_VEL
LIN {X 0,Y 516.966,Z 317.086,A -85,B 0,C 180,E1 -4941.4,E2 -4941.4} C_VEL
LIN {X 0,Y 517.009,Z 317.084,A -85,B 0,C 180,E1 -4943.757,E2 -4943.757} C_VEL
LIN {X 0,Y 517.083,Z 317.074,A -85,B 0,C 180,E1 -4947.663,E2 -4947.663} C_VEL
LIN {X 0,Y 517.091,Z 317.07,A -85,B 0,C 180,E1 -4950.779,E2 -4950.779} C_VEL
LIN {X 0,Y 517.01,Z 317.08,A -85,B 0,C 180,E1 -4953.117,E2 -4953.117} C_VEL
LIN {X 0,Y 517.008,Z 317.085,A -85,B 0,C 180,E1 -4956.243,E2 -4956.243} C_VEL
LIN {X 0,Y 516.95,Z 317.089,A -85,B 0,C 180,E1 -4959.389,E2 -4959.389} C_VEL
LIN {X 0,Y 516.95,Z 317.093,A -85,B 0,C 180,E1 -4961.808,E2 -4961.808} C_VEL
LIN {X 0,Y 516.943,Z 317.089,A -85,B 0,C 180,E1 -4965.147,E2 -4965.147} C_VEL
LIN {X 0,Y 516.924,Z 317.094,A -85,B 0,C 180,E1 -4968.222,E2 -4968.222} C_VEL
LIN {X 0,Y 516.911,Z 317.092,A -85,B 0,C 180,E1 -4970.702,E2 -4970.702} C_VEL
LIN {X 0,Y 516.91,Z 317.097,A -85,B 0,C 180,E1 -4974.072,E2 -4974.072} C_VEL
LIN {X 0,Y 516.925,Z 317.091,A -85,B 0,C 180,E1 -4976.658,E2 -4976.658} C_VEL
LIN {X 0,Y 516.91,Z 317.097,A -85,B 0,C 180,E1 -4979.524,E2 -4979.524} C_VEL
LIN {X 0,Y 516.897,Z 317.094,A -85,B 0,C 180,E1 -4982.544,E2 -4982.544} C_VEL
LIN {X 0,Y 516.881,Z 317.1,A -85,B 0,C 180,E1 -4985.333,E2 -4985.333} C_VEL
LIN {X 0,Y 516.881,Z 317.101,A -85,B 0,C 180,E1 -4987.944,E2 -4987.944} C_VEL
LIN {X 0,Y 516.883,Z 317.096,A -85,B 0,C 180,E1 -4990.742,E2 -4990.742} C_VEL
LIN {X 0,Y 516.882,Z 317.096,A -85,B 0,C 180,E1 -4992.832,E2 -4992.832} C_VEL
LIN {X 0,Y 516.895,Z 317.096,A -85,B 0,C 180,E1 -4995.008,E2 -4995.008} C_VEL
LIN {X 0,Y 516.914,Z 317.092,A -85,B 0,C 180,E1 -4998.399,E2 -4998.399} C_VEL
LIN {X 0,Y 516.881,Z 317.101,A -85,B 0,C 180,E1 -5001.285,E2 -5001.285} C_VEL
LIN {X 0,Y 516.872,Z 317.098,A -85,B 0,C 180,E1 -5004.22,E2 -5004.22} C_VEL
LIN {X 0,Y 516.883,Z 317.099,A -85,B 0,C 180,E1 -5007.053,E2 -5007.053} C_VEL
LIN {X 0,Y 516.889,Z 317.099,A -85,B 0,C 180,E1 -5009.797,E2 -5009.797} C_VEL
LIN {X 0,Y 516.927,Z 317.091,A -85,B 0,C 180,E1 -5012.468,E2 -5012.468} C_VEL
LIN {X 0,Y 516.909,Z 317.097,A -85,B 0,C 180,E1 -5015.072,E2 -5015.072} C_VEL
LIN {X 0,Y 516.904,Z 317.15,A -85,B 0,C 180,E1 -5016.996,E2 -5016.996} C_VEL
LIN {X 0,Y 518.973,Z 323.566,A -85,B 0,C 180,E1 -5017.154,E2 -5017.154} C_VEL
LIN {X 0,Y 518.559,Z 405.475,A -85,B 0,C 180,E1 -5018.353,E2 -5018.353} C_VEL
LIN {X 0,Y 518.4,Z 418.151,A -85,B 0,C 180,E1 -5018.685,E2 -5018.685} C_VEL
LIN {X 0,Y 518.224,Z 431.083,A -85,B 0,C 180,E1 -5019.198,E2 -5019.198} C_VEL
LIN {X 0,Y 518.033,Z 442.135,A -85,B 0,C 180,E1 -5019.784,E2 -5019.784} C_VEL
LIN {X 0,Y 517.752,Z 452.446,A -85,B 0,C 180,E1 -5020.473,E2 -5020.473} C_VEL
LIN {X 0,Y 517.525,Z 462.276,A -85,B 0,C 180,E1 -5021.287,E2 -5021.287} C_VEL
LIN {X 0,Y 517.248,Z 472.292,A -85,B 0,C 180,E1 -5022.315,E2 -5022.315} C_VEL
LIN {X 0,Y 517.005,Z 480.98,A -85,B 0,C 180,E1 -5023.414,E2 -5023.414} C_VEL
LIN {X 0,Y 516.795,Z 488.834,A -85,B 0,C 180,E1 -5024.663,E2 -5024.663} C_VEL
LIN {X 0,Y 516.638,Z 494.672,A -85,B 0,C 180,E1 -5025.827,E2 -5025.827} C_VEL
LIN {X 0,Y 516.521,Z 499.437,A -85,B 0,C 180,E1 -5027.027,E2 -5027.027} C_VEL
LIN {X 0,Y 516.481,Z 503.63,A -85,B 0,C 180,E1 -5028.449,E2 -5028.449} C_VEL
LIN {X 0,Y 516.375,Z 506.258,A -85,B 0,C 180,E1 -5029.809,E2 -5029.809} C_VEL
LIN {X 0,Y 516.402,Z 507.772,A -85,B 0,C 180,E1 -5031.391,E2 -5031.391} C_VEL
LIN {X 0,Y 516.407,Z 507.926,A -85,B 0,C 180,E1 -5032.178,E2 -5032.178} C_VEL
LIN {X 0,Y 516.433,Z 507.03,A -85,B 0,C 180,E1 -5033.75,E2 -5033.75} C_VEL
LIN {X 0,Y 516.465,Z 505.988,A -85,B 0,C 180,E1 -5034.534,E2 -5034.534} C_VEL
LIN {X 0,Y 516.504,Z 504.514,A -85,B 0,C 180,E1 -5035.317,E2 -5035.317} C_VEL
LIN {X 0,Y 516.56,Z 501.525,A -85,B 0,C 180,E1 -5036.49,E2 -5036.49} C_VEL
LIN {X 0,Y 516.609,Z 497.507,A -85,B 0,C 180,E1 -5037.661,E2 -5037.661} C_VEL
LIN {X 0,Y 516.764,Z 491.367,A -85,B 0,C 180,E1 -5039.026,E2 -5039.026} C_VEL
LIN {X 0,Y 516.982,Z 484.606,A -85,B 0,C 180,E1 -5040.195,E2 -5040.195} C_VEL
LIN {X 0,Y 517.192,Z 476.209,A -85,B 0,C 180,E1 -5041.363,E2 -5041.363} C_VEL
LIN {X 0,Y 517.445,Z 467.595,A -85,B 0,C 180,E1 -5042.336,E2 -5042.336} C_VEL
LIN {X 0,Y 517.715,Z 458.096,A -85,B 0,C 180,E1 -5043.21,E2 -5043.21} C_VEL
LIN {X 0,Y 517.935,Z 447.653,A -85,B 0,C 180,E1 -5043.988,E2 -5043.988} C_VEL
LIN {X 0,Y 518.202,Z 436.09,A -85,B 0,C 180,E1 -5044.668,E2 -5044.668} C_VEL
LIN {X 0,Y 518.338,Z 424.145,A -85,B 0,C 180,E1 -5045.203,E2 -5045.203} C_VEL
LIN {X 0,Y 518.447,Z 410.859,A -85,B 0,C 180,E1 -5045.616,E2 -5045.616} C_VEL
LIN {X 0,Y 518.574,Z 396.258,A -85,B 0,C 180,E1 -5045.883,E2 -5045.883} C_VEL
LIN {X 0,Y 518.89,Z 323.253,A -85,B 0,C 180,E1 -5046.945,E2 -5046.945} C_VEL
LIN {X 0,Y 516.959,Z 317.092,A -85,B 0,C 180,E1 -5047.115,E2 -5047.115} C_VEL
LIN {X 0,Y 516.86,Z 317.105,A -85,B 0,C 180,E1 -5050.182,E2 -5050.182} C_VEL
LIN {X 0,Y 516.887,Z 317.103,A -85,B 0,C 180,E1 -5052.565,E2 -5052.565} C_VEL
LIN {X 0,Y 516.942,Z 317.091,A -85,B 0,C 180,E1 -5055.143,E2 -5055.143} C_VEL
LIN {X 0,Y 516.854,Z 317.108,A -85,B 0,C 180,E1 -5058.225,E2 -5058.225} C_VEL
LIN {X 0,Y 516.866,Z 317.104,A -85,B 0,C 180,E1 -5060.704,E2 -5060.704} C_VEL
LIN {X 0,Y 516.854,Z 317.099,A -85,B 0,C 180,E1 -5063.225,E2 -5063.225} C_VEL
LIN {X 0,Y 516.863,Z 317.106,A -85,B 0,C 180,E1 -5066.177,E2 -5066.177} C_VEL
LIN {X 0,Y 516.907,Z 317.093,A -85,B 0,C 180,E1 -5069.306,E2 -5069.306} C_VEL
LIN {X 0,Y 516.896,Z 317.097,A -85,B 0,C 180,E1 -5072.542,E2 -5072.542} C_VEL
LIN {X 0,Y 516.854,Z 317.098,A -85,B 0,C 180,E1 -5075.327,E2 -5075.327} C_VEL
LIN {X 0,Y 516.877,Z 317.096,A -85,B 0,C 180,E1 -5078.717,E2 -5078.717} C_VEL
LIN {X 0,Y 516.853,Z 317.104,A -85,B 0,C 180,E1 -5081.782,E2 -5081.782} C_VEL
LIN {X 0,Y 516.9,Z 317.094,A -85,B 0,C 180,E1 -5085.007,E2 -5085.007} C_VEL
LIN {X 0,Y 516.891,Z 317.096,A -85,B 0,C 180,E1 -5088.402,E2 -5088.402} C_VEL
LIN {X 0,Y 516.88,Z 317.1,A -85,B 0,C 180,E1 -5091.284,E2 -5091.284} C_VEL
LIN {X 0,Y 516.868,Z 317.1,A -85,B 0,C 180,E1 -5094.219,E2 -5094.219} C_VEL
LIN {X 0,Y 516.885,Z 317.098,A -85,B 0,C 180,E1 -5097.052,E2 -5097.052} C_VEL
LIN {X 0,Y 516.896,Z 317.1,A -85,B 0,C 180,E1 -5099.796,E2 -5099.796} C_VEL
LIN {X 0,Y 516.924,Z 317.111,A -85,B 0,C 180,E1 -5101.757,E2 -5101.757} C_VEL
LIN {X 0,Y 519.505,Z 329.332,A -85,B 0,C 180,E1 -5103.485,E2 -5103.485} C_VEL
LIN {X 0,Y 519.009,Z 349.206,A -85,B 0,C 180,E1 -5106.031,E2 -5106.031} C_VEL
LIN {X 0,Y 518.446,Z 372.575,A -85,B 0,C 180,E1 -5108.988,E2 -5108.988} C_VEL
LIN {X 0,Y 517.85,Z 398.717,A -85,B 0,C 180,E1 -5112.22,E2 -5112.22} C_VEL
LIN {X 0,Y 517.413,Z 418.362,A -85,B 0,C 180,E1 -5114.629,E2 -5114.629} C_VEL
LIN {X 0,Y 518.99,Z 431.753,A -85,B 0,C 180,E1 -5114.884,E2 -5114.884} C_VEL
LIN {X 0,Y 518.5,Z 524.54,A -85,B 0,C 180,E1 -5116.203,E2 -5116.203} C_VEL
LIN {X 0,Y 518.287,Z 537.802,A -85,B 0,C 180,E1 -5116.497,E2 -5116.497} C_VEL
LIN {X 0,Y 518.068,Z 549.971,A -85,B 0,C 180,E1 -5116.916,E2 -5116.916} C_VEL
LIN {X 0,Y 517.759,Z 561.466,A -85,B 0,C 180,E1 -5117.456,E2 -5117.456} C_VEL
LIN {X 0,Y 517.499,Z 572.866,A -85,B 0,C 180,E1 -5118.149,E2 -5118.149} C_VEL
LIN {X 0,Y 517.215,Z 584.438,A -85,B 0,C 180,E1 -5119.033,E2 -5119.033} C_VEL
LIN {X 0,Y 516.931,Z 594.685,A -85,B 0,C 180,E1 -5120.017,E2 -5120.017} C_VEL
LIN {X 0,Y 516.712,Z 604.597,A -85,B 0,C 180,E1 -5121.198,E2 -5121.198} C_VEL
LIN {X 0,Y 516.555,Z 612.518,A -85,B 0,C 180,E1 -5122.377,E2 -5122.377} C_VEL
LIN {X 0,Y 516.438,Z 618.276,A -85,B 0,C 180,E1 -5123.43,E2 -5123.43} C_VEL
LIN {X 0,Y 516.4,Z 623.174,A -85,B 0,C 180,E1 -5124.533,E2 -5124.533} C_VEL
LIN {X 0,Y 516.367,Z 627.245,A -85,B 0,C 180,E1 -5125.707,E2 -5125.707} C_VEL
LIN {X 0,Y 516.339,Z 630.246,A -85,B 0,C 180,E1 -5126.879,E2 -5126.879} C_VEL
LIN {X 0,Y 516.281,Z 631.671,A -85,B 0,C 180,E1 -5127.659,E2 -5127.659} C_VEL
LIN {X 0,Y 516.221,Z 633.301,A -85,B 0,C 180,E1 -5129.22,E2 -5129.22} C_VEL
LIN {X 0,Y 516.223,Z 633.512,A -85,B 0,C 180,E1 -5130,E2 -5130} C_VEL
LIN {X 0,Y 516.223,Z 633.282,A -85,B 0,C 180,E1 -5130.78,E2 -5130.78} C_VEL
LIN {X 0,Y 516.286,Z 631.625,A -85,B 0,C 180,E1 -5132.34,E2 -5132.34} C_VEL
LIN {X 0,Y 516.339,Z 630.172,A -85,B 0,C 180,E1 -5133.121,E2 -5133.121} C_VEL
LIN {X 0,Y 516.366,Z 627.131,A -85,B 0,C 180,E1 -5134.293,E2 -5134.293} C_VEL
LIN {X 0,Y 516.4,Z 623.013,A -85,B 0,C 180,E1 -5135.467,E2 -5135.467} C_VEL
LIN {X 0,Y 516.489,Z 616.816,A -85,B 0,C 180,E1 -5136.812,E2 -5136.812} C_VEL
LIN {X 0,Y 516.598,Z 609.766,A -85,B 0,C 180,E1 -5138.016,E2 -5138.016} C_VEL
LIN {X 0,Y 516.77,Z 601.164,A -85,B 0,C 180,E1 -5139.195,E2 -5139.195} C_VEL
LIN {X 0,Y 517.02,Z 591.326,A -85,B 0,C 180,E1 -5140.277,E2 -5140.277} C_VEL
LIN {X 0,Y 517.286,Z 580.216,A -85,B 0,C 180,E1 -5141.262,E2 -5141.262} C_VEL
LIN {X 0,Y 517.491,Z 569.34,A -85,B 0,C 180,E1 -5142.035,E2 -5142.035} C_VEL
LIN {X 0,Y 517.798,Z 557.602,A -85,B 0,C 180,E1 -5142.692,E2 -5142.692} C_VEL
LIN {X 0,Y 518.038,Z 544.834,A -85,B 0,C 180,E1 -5143.234,E2 -5143.234} C_VEL
LIN {X 0,Y 518.332,Z 531.46,A -85,B 0,C 180,E1 -5143.626,E2 -5143.626} C_VEL
LIN {X 0,Y 518.551,Z 512.238,A -85,B 0,C 180,E1 -5143.945,E2 -5143.945} C_VEL
LIN {X 0,Y 518.811,Z 430.084,A -85,B 0,C 180,E1 -5145.122,E2 -5145.122} C_VEL
LIN {X 0,Y 517.387,Z 416.777,A -85,B 0,C 180,E1 -5145.374,E2 -5145.374} C_VEL
LIN {X 0,Y 517.839,Z 388.329,A -85,B 0,C 180,E1 -5148.804,E2 -5148.804} C_VEL
LIN {X 0,Y 518.255,Z 364.749,A -85,B 0,C 180,E1 -5151.687,E2 -5151.687} C_VEL
LIN {X 0,Y 518.706,Z 342.909,A -85,B 0,C 180,E1 -5154.409,E2 -5154.409} C_VEL
LIN {X 0,Y 518.932,Z 327.852,A -85,B 0,C 180,E1 -5156.33,E2 -5156.33} C_VEL
LIN {X 0,Y 516.885,Z 317.102,A -85,B 0,C 180,E1 -5157.839,E2 -5157.839} C_VEL
LIN {X 0,Y 516.895,Z 317.103,A -85,B 0,C 180,E1 -5160.204,E2 -5160.204} C_VEL
LIN {X 0,Y 516.884,Z 317.1,A -85,B 0,C 180,E1 -5162.948,E2 -5162.948} C_VEL
LIN {X 0,Y 516.871,Z 317.101,A -85,B 0,C 180,E1 -5165.78,E2 -5165.78} C_VEL
LIN {X 0,Y 516.879,Z 317.101,A -85,B 0,C 180,E1 -5168.716,E2 -5168.716} C_VEL
LIN {X 0,Y 516.886,Z 317.1,A -85,B 0,C 180,E1 -5171.778,E2 -5171.778} C_VEL
LIN {X 0,Y 516.898,Z 317.095,A -85,B 0,C 180,E1 -5175.007,E2 -5175.007} C_VEL
LIN {X 0,Y 516.888,Z 317.1,A -85,B 0,C 180,E1 -5178.402,E2 -5178.402} C_VEL
LIN {X 0,Y 516.875,Z 317.097,A -85,B 0,C 180,E1 -5181.283,E2 -5181.283} C_VEL
LIN {X 0,Y 516.852,Z 317.1,A -85,B 0,C 180,E1 -5184.673,E2 -5184.673} C_VEL
LIN {X 0,Y 516.894,Z 317.097,A -85,B 0,C 180,E1 -5187.457,E2 -5187.457} C_VEL
LIN {X 0,Y 516.905,Z 317.094,A -85,B 0,C 180,E1 -5190.694,E2 -5190.694} C_VEL
LIN {X 0,Y 516.861,Z 317.106,A -85,B 0,C 180,E1 -5193.823,E2 -5193.823} C_VEL
LIN {X 0,Y 516.852,Z 317.102,A -85,B 0,C 180,E1 -5196.775,E2 -5196.775} C_VEL
LIN {X 0,Y 516.876,Z 317.103,A -85,B 0,C 180,E1 -5199.752,E2 -5199.752} C_VEL
LIN {X 0,Y 516.886,Z 317.097,A -85,B 0,C 180,E1 -5202.594,E2 -5202.594} C_VEL
LIN {X 0,Y 516.935,Z 317.096,A -85,B 0,C 180,E1 -5205.03,E2 -5205.03} C_VEL
LIN {X 0,Y 516.917,Z 317.099,A -85,B 0,C 180,E1 -5206.985,E2 -5206.985} C_VEL
LIN {X 0,Y 519.009,Z 323.691,A -85,B 0,C 180,E1 -5207.153,E2 -5207.153} C_VEL
LIN {X 0,Y 518.45,Z 406.82,A -85,B 0,C 180,E1 -5208.391,E2 -5208.391} C_VEL
LIN {X 0,Y 518.385,Z 419.602,A -85,B 0,C 180,E1 -5208.737,E2 -5208.737} C_VEL
LIN {X 0,Y 518.236,Z 432.562,A -85,B 0,C 180,E1 -5209.253,E2 -5209.253} C_VEL
LIN {X 0,Y 518.047,Z 443.489,A -85,B 0,C 180,E1 -5209.842,E2 -5209.842} C_VEL
LIN {X 0,Y 517.763,Z 454.865,A -85,B 0,C 180,E1 -5210.625,E2 -5210.625} C_VEL
LIN {X 0,Y 517.531,Z 465.081,A -85,B 0,C 180,E1 -5211.507,E2 -5211.507} C_VEL
LIN {X 0,Y 517.258,Z 474.003,A -85,B 0,C 180,E1 -5212.455,E2 -5212.455} C_VEL
LIN {X 0,Y 517.005,Z 482.566,A -85,B 0,C 180,E1 -5213.582,E2 -5213.582} C_VEL
LIN {X 0,Y 516.937,Z 489.613,A -85,B 0,C 180,E1 -5214.734,E2 -5214.734} C_VEL
LIN {X 0,Y 516.729,Z 494.504,A -85,B 0,C 180,E1 -5215.71,E2 -5215.71} C_VEL
LIN {X 0,Y 516.564,Z 499.227,A -85,B 0,C 180,E1 -5216.88,E2 -5216.88} C_VEL
LIN {X 0,Y 516.559,Z 502.833,A -85,B 0,C 180,E1 -5218.05,E2 -5218.05} C_VEL
LIN {X 0,Y 516.399,Z 505.462,A -85,B 0,C 180,E1 -5219.22,E2 -5219.22} C_VEL
LIN {X 0,Y 516.381,Z 506.69,A -85,B 0,C 180,E1 -5220,E2 -5220} C_VEL
LIN {X 0,Y 516.386,Z 507.517,A -85,B 0,C 180,E1 -5220.779,E2 -5220.779} C_VEL
LIN {X 0,Y 516.329,Z 507.931,A -85,B 0,C 180,E1 -5221.56,E2 -5221.56} C_VEL
LIN {X 0,Y 516.431,Z 507.573,A -85,B 0,C 180,E1 -5223.12,E2 -5223.12} C_VEL
LIN {X 0,Y 516.429,Z 506.807,A -85,B 0,C 180,E1 -5223.901,E2 -5223.901} C_VEL
LIN {X 0,Y 516.498,Z 504.059,A -85,B 0,C 180,E1 -5225.465,E2 -5225.465} C_VEL
LIN {X 0,Y 516.578,Z 500.665,A -85,B 0,C 180,E1 -5226.704,E2 -5226.704} C_VEL
LIN {X 0,Y 516.648,Z 496.61,A -85,B 0,C 180,E1 -5227.818,E2 -5227.818} C_VEL
LIN {X 0,Y 516.772,Z 491.153,A -85,B 0,C 180,E1 -5228.997,E2 -5228.997} C_VEL
LIN {X 0,Y 516.93,Z 484.311,A -85,B 0,C 180,E1 -5230.18,E2 -5230.18} C_VEL
LIN {X 0,Y 517.1,Z 477.303,A -85,B 0,C 180,E1 -5231.167,E2 -5231.167} C_VEL
LIN {X 0,Y 517.342,Z 468.822,A -85,B 0,C 180,E1 -5232.155,E2 -5232.155} C_VEL
LIN {X 0,Y 517.607,Z 458.296,A -85,B 0,C 180,E1 -5233.145,E2 -5233.145} C_VEL
LIN {X 0,Y 517.845,Z 447.818,A -85,B 0,C 180,E1 -5233.939,E2 -5233.939} C_VEL
LIN {X 0,Y 518.139,Z 436.219,A -85,B 0,C 180,E1 -5234.633,E2 -5234.633} C_VEL
LIN {X 0,Y 518.356,Z 423.404,A -85,B 0,C 180,E1 -5235.208,E2 -5235.208} C_VEL
LIN {X 0,Y 518.481,Z 410.207,A -85,B 0,C 180,E1 -5235.626,E2 -5235.626} C_VEL
LIN {X 0,Y 518.564,Z 395.952,A -85,B 0,C 180,E1 -5235.89,E2 -5235.89} C_VEL
LIN {X 0,Y 518.912,Z 323.443,A -85,B 0,C 180,E1 -5236.94,E2 -5236.94} C_VEL
LIN {X 0,Y 516.941,Z 317.094,A -85,B 0,C 180,E1 -5237.11,E2 -5237.11} C_VEL
LIN {X 0,Y 516.941,Z 317.092,A -85,B 0,C 180,E1 -5240.268,E2 -5240.268} C_VEL
LIN {X 0,Y 516.865,Z 317.099,A -85,B 0,C 180,E1 -5243.223,E2 -5243.223} C_VEL
LIN {X 0,Y 516.943,Z 317.091,A -85,B 0,C 180,E1 -5246.195,E2 -5246.195} C_VEL
LIN {X 0,Y 516.921,Z 317.091,A -85,B 0,C 180,E1 -5249.304,E2 -5249.304} C_VEL
LIN {X 0,Y 516.894,Z 317.101,A -85,B 0,C 180,E1 -5252.543,E2 -5252.543} C_VEL
LIN {X 0,Y 516.865,Z 317.098,A -85,B 0,C 180,E1 -5255.329,E2 -5255.329} C_VEL
LIN {X 0,Y 516.879,Z 317.098,A -85,B 0,C 180,E1 -5257.943,E2 -5257.943} C_VEL
LIN {X 0,Y 516.87,Z 317.101,A -85,B 0,C 180,E1 -5258.487,E2 -5258.487} C_VEL
LIN {X 0,Y 516.23,Z 317.184,A -85,B 0,C 180,E1 -5259.138,E2 -5259.138} C_VEL
LIN {X 0,Y 513.413,Z 317.533,A -85,B 0,C 180,E1 -5260.195,E2 -5260.195} C_VEL
LIN {X 0,Y 511.004,Z 317.83,A -85,B 0,C 180,E1 -5261.046,E2 -5261.046} C_VEL
LIN {X 0,Y 509.949,Z 317.96,A -85,B 0,C 180,E1 -5261.703,E2 -5261.703} C_VEL
LIN {X 0,Y 509.852,Z 317.973,A -85,B 0,C 180,E1 -5261.926,E2 -5261.926} C_VEL
LIN {X 0,Y 509.837,Z 317.973,A -85,B 0,C 180,E1 -5265.33,E2 -5265.33} C_VEL
LIN {X 0,Y 509.853,Z 317.978,A -85,B 0,C 180,E1 -5268.574,E2 -5268.574} C_VEL
LIN {X 0,Y 509.85,Z 317.973,A -85,B 0,C 180,E1 -5271.786,E2 -5271.786} C_VEL
LIN {X 0,Y 509.843,Z 317.978,A -85,B 0,C 180,E1 -5274.623,E2 -5274.623} C_VEL
LIN {X 0,Y 509.861,Z 317.971,A -85,B 0,C 180,E1 -5277.481,E2 -5277.481} C_VEL
LIN {X 0,Y 509.856,Z 317.978,A -85,B 0,C 180,E1 -5280.273,E2 -5280.273} C_VEL
LIN {X 0,Y 509.883,Z 317.969,A -85,B 0,C 180,E1 -5282.944,E2 -5282.944} C_VEL
LIN {X 0,Y 509.868,Z 317.971,A -85,B 0,C 180,E1 -5285.574,E2 -5285.574} C_VEL
LIN {X 0,Y 509.848,Z 317.972,A -85,B 0,C 180,E1 -5288.998,E2 -5288.998} C_VEL
LIN {X 0,Y 509.886,Z 317.972,A -85,B 0,C 180,E1 -5291.999,E2 -5291.999} C_VEL
LIN {X 0,Y 509.908,Z 317.966,A -85,B 0,C 180,E1 -5294.819,E2 -5294.819} C_VEL
LIN {X 0,Y 509.899,Z 317.973,A -85,B 0,C 180,E1 -5298.124,E2 -5298.124} C_VEL
LIN {X 0,Y 509.913,Z 317.964,A -85,B 0,C 180,E1 -5301.28,E2 -5301.28} C_VEL
LIN {X 0,Y 509.977,Z 317.959,A -85,B 0,C 180,E1 -5303.67,E2 -5303.67} C_VEL
LIN {X 0,Y 510.054,Z 317.95,A -85,B 0,C 180,E1 -5307.631,E2 -5307.631} C_VEL
LIN {X 0,Y 510.062,Z 317.946,A -85,B 0,C 180,E1 -5310.79,E2 -5310.79} C_VEL
LIN {X 0,Y 509.953,Z 317.959,A -85,B 0,C 180,E1 -5313.16,E2 -5313.16} C_VEL
LIN {X 0,Y 509.977,Z 317.96,A -85,B 0,C 180,E1 -5316.33,E2 -5316.33} C_VEL
LIN {X 0,Y 509.913,Z 317.965,A -85,B 0,C 180,E1 -5318.72,E2 -5318.72} C_VEL
LIN {X 0,Y 509.902,Z 317.973,A -85,B 0,C 180,E1 -5321.932,E2 -5321.932} C_VEL
LIN {X 0,Y 509.892,Z 317.968,A -85,B 0,C 180,E1 -5325.242,E2 -5325.242} C_VEL
LIN {X 0,Y 509.887,Z 317.974,A -85,B 0,C 180,E1 -5328.001,E2 -5328.001} C_VEL
LIN {X 0,Y 509.849,Z 317.972,A -85,B 0,C 180,E1 -5331.002,E2 -5331.002} C_VEL
LIN {X 0,Y 509.836,Z 317.978,A -85,B 0,C 180,E1 -5333.563,E2 -5333.563} C_VEL
LIN {X 0,Y 509.911,Z 317.966,A -85,B 0,C 180,E1 -5336.379,E2 -5336.379} C_VEL
LIN {X 0,Y 509.876,Z 317.969,A -85,B 0,C 180,E1 -5338.845,E2 -5338.845} C_VEL
LIN {X 0,Y 509.821,Z 317.981,A -85,B 0,C 180,E1 -5341.59,E2 -5341.59} C_VEL
LIN {X 0,Y 509.853,Z 317.972,A -85,B 0,C 180,E1 -5344.414,E2 -5344.414} C_VEL
LIN {X 0,Y 509.819,Z 317.98,A -85,B 0,C 180,E1 -5347.341,E2 -5347.341} C_VEL
LIN {X 0,Y 509.838,Z 317.974,A -85,B 0,C 180,E1 -5350.383,E2 -5350.383} C_VEL
LIN {X 0,Y 509.823,Z 317.978,A -85,B 0,C 180,E1 -5353.063,E2 -5353.063} C_VEL
LIN {X 0,Y 509.824,Z 317.981,A -85,B 0,C 180,E1 -5355.794,E2 -5355.794} C_VEL
LIN {X 0,Y 509.856,Z 317.971,A -85,B 0,C 180,E1 -5358.575,E2 -5358.575} C_VEL
LIN {X 0,Y 509.852,Z 317.977,A -85,B 0,C 180,E1 -5361.787,E2 -5361.787} C_VEL
LIN {X 0,Y 509.831,Z 317.975,A -85,B 0,C 180,E1 -5364.623,E2 -5364.623} C_VEL
LIN {X 0,Y 509.862,Z 317.977,A -85,B 0,C 180,E1 -5367.481,E2 -5367.481} C_VEL
LIN {X 0,Y 509.86,Z 317.971,A -85,B 0,C 180,E1 -5370.274,E2 -5370.274} C_VEL
LIN {X 0,Y 509.885,Z 317.971,A -85,B 0,C 180,E1 -5372.945,E2 -5372.945} C_VEL
LIN {X 0,Y 509.865,Z 317.977,A -85,B 0,C 180,E1 -5375.574,E2 -5375.574} C_VEL
LIN {X 0,Y 509.849,Z 317.975,A -85,B 0,C 180,E1 -5376.777,E2 -5376.777} C_VEL
LIN {X 0,Y 512.163,Z 325.856,A -85,B 0,C 180,E1 -5376.983,E2 -5376.983} C_VEL
LIN {X 0,Y 511.658,Z 406.05,A -85,B 0,C 180,E1 -5378.178,E2 -5378.178} C_VEL
LIN {X 0,Y 511.493,Z 418.773,A -85,B 0,C 180,E1 -5378.515,E2 -5378.515} C_VEL
LIN {X 0,Y 511.337,Z 431.209,A -85,B 0,C 180,E1 -5379.01,E2 -5379.01} C_VEL
LIN {X 0,Y 511.111,Z 442.98,A -85,B 0,C 180,E1 -5379.638,E2 -5379.638} C_VEL
LIN {X 0,Y 510.803,Z 454.206,A -85,B 0,C 180,E1 -5380.405,E2 -5380.405} C_VEL
LIN {X 0,Y 510.525,Z 464.898,A -85,B 0,C 180,E1 -5381.334,E2 -5381.334} C_VEL
LIN {X 0,Y 510.231,Z 474.491,A -85,B 0,C 180,E1 -5382.361,E2 -5382.361} C_VEL
LIN {X 0,Y 510.002,Z 482.302,A -85,B 0,C 180,E1 -5383.385,E2 -5383.385} C_VEL
LIN {X 0,Y 509.803,Z 489.84,A -85,B 0,C 180,E1 -5384.611,E2 -5384.611} C_VEL
LIN {X 0,Y 509.606,Z 496.736,A -85,B 0,C 180,E1 -5386.035,E2 -5386.035} C_VEL
LIN {X 0,Y 509.505,Z 501.217,A -85,B 0,C 180,E1 -5387.25,E2 -5387.25} C_VEL
LIN {X 0,Y 509.455,Z 504.363,A -85,B 0,C 180,E1 -5388.368,E2 -5388.368} C_VEL
LIN {X 0,Y 509.346,Z 506.922,A -85,B 0,C 180,E1 -5389.667,E2 -5389.667} C_VEL
LIN {X 0,Y 509.376,Z 508.561,A -85,B 0,C 180,E1 -5391.271,E2 -5391.271} C_VEL
LIN {X 0,Y 509.374,Z 508.79,A -85,B 0,C 180,E1 -5392.07,E2 -5392.07} C_VEL
LIN {X 0,Y 509.396,Z 507.992,A -85,B 0,C 180,E1 -5393.664,E2 -5393.664} C_VEL
LIN {X 0,Y 509.444,Z 507.016,A -85,B 0,C 180,E1 -5394.459,E2 -5394.459} C_VEL
LIN {X 0,Y 509.486,Z 505.598,A -85,B 0,C 180,E1 -5395.253,E2 -5395.253} C_VEL
LIN {X 0,Y 509.525,Z 502.699,A -85,B 0,C 180,E1 -5396.442,E2 -5396.442} C_VEL
LIN {X 0,Y 509.594,Z 498.767,A -85,B 0,C 180,E1 -5397.629,E2 -5397.629} C_VEL
LIN {X 0,Y 509.694,Z 493.689,A -85,B 0,C 180,E1 -5398.815,E2 -5398.815} C_VEL
LIN {X 0,Y 509.957,Z 487.288,A -85,B 0,C 180,E1 -5400,E2 -5400} C_VEL
LIN {X 0,Y 510.171,Z 479.364,A -85,B 0,C 180,E1 -5401.184,E2 -5401.184} C_VEL
LIN {X 0,Y 510.407,Z 471.196,A -85,B 0,C 180,E1 -5402.17,E2 -5402.17} C_VEL
LIN {X 0,Y 510.697,Z 461.167,A -85,B 0,C 180,E1 -5403.156,E2 -5403.156} C_VEL
LIN {X 0,Y 510.934,Z 451.285,A -85,B 0,C 180,E1 -5403.944,E2 -5403.944} C_VEL
LIN {X 0,Y 511.193,Z 440.486,A -85,B 0,C 180,E1 -5404.633,E2 -5404.633} C_VEL
LIN {X 0,Y 511.392,Z 428.407,A -85,B 0,C 180,E1 -5405.224,E2 -5405.224} C_VEL
LIN {X 0,Y 511.536,Z 415.981,A -85,B 0,C 180,E1 -5405.668,E2 -5405.668} C_VEL
LIN {X 0,Y 511.618,Z 403.035,A -85,B 0,C 180,E1 -5405.963,E2 -5405.963} C_VEL
LIN {X 0,Y 512.181,Z 325.381,A -85,B 0,C 180,E1 -5407.119,E2 -5407.119} C_VEL
LIN {X 0,Y 509.894,Z 317.971,A -85,B 0,C 180,E1 -5407.323,E2 -5407.323} C_VEL
LIN {X 0,Y 509.814,Z 317.984,A -85,B 0,C 180,E1 -5410.324,E2 -5410.324} C_VEL
LIN {X 0,Y 509.849,Z 317.979,A -85,B 0,C 180,E1 -5412.742,E2 -5412.742} C_VEL
LIN {X 0,Y 509.9,Z 317.968,A -85,B 0,C 180,E1 -5415.242,E2 -5415.242} C_VEL
LIN {X 0,Y 509.816,Z 317.984,A -85,B 0,C 180,E1 -5418.486,E2 -5418.486} C_VEL
LIN {X 0,Y 509.815,Z 317.98,A -85,B 0,C 180,E1 -5421.004,E2 -5421.004} C_VEL
LIN {X 0,Y 509.813,Z 317.977,A -85,B 0,C 180,E1 -5423.565,E2 -5423.565} C_VEL
LIN {X 0,Y 509.803,Z 317.986,A -85,B 0,C 180,E1 -5426.353,E2 -5426.353} C_VEL
LIN {X 0,Y 509.837,Z 317.975,A -85,B 0,C 180,E1 -5428.847,E2 -5428.847} C_VEL
LIN {X 0,Y 509.815,Z 317.979,A -85,B 0,C 180,E1 -5431.591,E2 -5431.591} C_VEL
LIN {X 0,Y 509.837,Z 317.976,A -85,B 0,C 180,E1 -5434.415,E2 -5434.415} C_VEL
LIN {X 0,Y 509.784,Z 317.98,A -85,B 0,C 180,E1 -5437.344,E2 -5437.344} C_VEL
LIN {X 0,Y 509.817,Z 317.977,A -85,B 0,C 180,E1 -5440.385,E2 -5440.385} C_VEL
LIN {X 0,Y 509.81,Z 317.98,A -85,B 0,C 180,E1 -5443.573,E2 -5443.573} C_VEL
LIN {X 0,Y 509.811,Z 317.978,A -85,B 0,C 180,E1 -5446.427,E2 -5446.427} C_VEL
LIN {X 0,Y 509.816,Z 317.979,A -85,B 0,C 180,E1 -5449.306,E2 -5449.306} C_VEL
LIN {X 0,Y 509.852,Z 317.979,A -85,B 0,C 180,E1 -5451.787,E2 -5451.787} C_VEL
LIN {X 0,Y 509.829,Z 317.975,A -85,B 0,C 180,E1 -5454.621,E2 -5454.621} C_VEL
LIN {X 0,Y 509.864,Z 317.978,A -85,B 0,C 180,E1 -5457.481,E2 -5457.481} C_VEL
LIN {X 0,Y 509.863,Z 317.974,A -85,B 0,C 180,E1 -5460.274,E2 -5460.274} C_VEL
LIN {X 0,Y 509.886,Z 318.078,A -85,B 0,C 180,E1 -5461.549,E2 -5461.549} C_VEL
LIN {X 0,Y 512.646,Z 330.978,A -85,B 0,C 180,E1 -5463.402,E2 -5463.402} C_VEL
LIN {X 0,Y 512.09,Z 350.211,A -85,B 0,C 180,E1 -5465.902,E2 -5465.902} C_VEL
LIN {X 0,Y 511.4,Z 374.889,A -85,B 0,C 180,E1 -5469.065,E2 -5469.065} C_VEL
LIN {X 0,Y 510.834,Z 399.895,A -85,B 0,C 180,E1 -5472.2,E2 -5472.2} C_VEL
LIN {X 0,Y 510.402,Z 417.64,A -85,B 0,C 180,E1 -5474.414,E2 -5474.414} C_VEL
LIN {X 0,Y 512.096,Z 431.932,A -85,B 0,C 180,E1 -5474.691,E2 -5474.691} C_VEL
LIN {X 0,Y 511.551,Z 525.69,A -85,B 0,C 180,E1 -5476.063,E2 -5476.063} C_VEL
LIN {X 0,Y 511.314,Z 538.954,A -85,B 0,C 180,E1 -5476.386,E2 -5476.386} C_VEL
LIN {X 0,Y 511.021,Z 552.2,A -85,B 0,C 180,E1 -5476.884,E2 -5476.884} C_VEL
LIN {X 0,Y 510.709,Z 563.472,A -85,B 0,C 180,E1 -5477.457,E2 -5477.457} C_VEL
LIN {X 0,Y 510.438,Z 574.655,A -85,B 0,C 180,E1 -5478.182,E2 -5478.182} C_VEL
LIN {X 0,Y 510.141,Z 585.653,A -85,B 0,C 180,E1 -5479.08,E2 -5479.08} C_VEL
LIN {X 0,Y 509.847,Z 595.546,A -85,B 0,C 180,E1 -5480.078,E2 -5480.078} C_VEL
LIN {X 0,Y 509.653,Z 603.669,A -85,B 0,C 180,E1 -5481.075,E2 -5481.075} C_VEL
LIN {X 0,Y 509.476,Z 611.622,A -85,B 0,C 180,E1 -5482.27,E2 -5482.27} C_VEL
LIN {X 0,Y 509.35,Z 617.888,A -85,B 0,C 180,E1 -5483.443,E2 -5483.443} C_VEL
LIN {X 0,Y 509.34,Z 622.312,A -85,B 0,C 180,E1 -5484.457,E2 -5484.457} C_VEL
LIN {X 0,Y 509.297,Z 626.392,A -85,B 0,C 180,E1 -5485.647,E2 -5485.647} C_VEL
LIN {X 0,Y 509.284,Z 629.401,A -85,B 0,C 180,E1 -5486.836,E2 -5486.836} C_VEL
LIN {X 0,Y 509.225,Z 630.829,A -85,B 0,C 180,E1 -5487.627,E2 -5487.627} C_VEL
LIN {X 0,Y 509.183,Z 631.842,A -85,B 0,C 180,E1 -5488.418,E2 -5488.418} C_VEL
LIN {X 0,Y 509.17,Z 632.455,A -85,B 0,C 180,E1 -5489.209,E2 -5489.209} C_VEL
LIN {X 0,Y 509.175,Z 632.662,A -85,B 0,C 180,E1 -5490,E2 -5490} C_VEL
LIN {X 0,Y 509.174,Z 632.426,A -85,B 0,C 180,E1 -5490.791,E2 -5490.791} C_VEL
LIN {X 0,Y 509.189,Z 631.788,A -85,B 0,C 180,E1 -5491.582,E2 -5491.582} C_VEL
LIN {X 0,Y 509.233,Z 630.745,A -85,B 0,C 180,E1 -5492.373,E2 -5492.373} C_VEL
LIN {X 0,Y 509.285,Z 629.279,A -85,B 0,C 180,E1 -5493.164,E2 -5493.164} C_VEL
LIN {X 0,Y 509.301,Z 626.212,A -85,B 0,C 180,E1 -5494.353,E2 -5494.353} C_VEL
LIN {X 0,Y 509.341,Z 622.064,A -85,B 0,C 180,E1 -5495.543,E2 -5495.543} C_VEL
LIN {X 0,Y 509.418,Z 616.049,A -85,B 0,C 180,E1 -5496.864,E2 -5496.864} C_VEL
LIN {X 0,Y 509.546,Z 608.725,A -85,B 0,C 180,E1 -5498.127,E2 -5498.127} C_VEL
LIN {X 0,Y 509.711,Z 600.064,A -85,B 0,C 180,E1 -5499.324,E2 -5499.324} C_VEL
LIN {X 0,Y 509.963,Z 590.161,A -85,B 0,C 180,E1 -5500.421,E2 -5500.421} C_VEL
LIN {X 0,Y 510.264,Z 578.975,A -85,B 0,C 180,E1 -5501.419,E2 -5501.419} C_VEL
LIN {X 0,Y 510.521,Z 567.3,A -85,B 0,C 180,E1 -5502.246,E2 -5502.246} C_VEL
LIN {X 0,Y 510.818,Z 555.114,A -85,B 0,C 180,E1 -5502.919,E2 -5502.919} C_VEL
LIN {X 0,Y 511.116,Z 543.224,A -85,B 0,C 180,E1 -5503.417,E2 -5503.417} C_VEL
LIN {X 0,Y 511.342,Z 530.521,A -85,B 0,C 180,E1 -5503.791,E2 -5503.791} C_VEL
LIN {X 0,Y 511.603,Z 511.379,A -85,B 0,C 180,E1 -5504.113,E2 -5504.113} C_VEL
LIN {X 0,Y 511.914,Z 430.671,A -85,B 0,C 180,E1 -5505.303,E2 -5505.303} C_VEL
LIN {X 0,Y 510.297,Z 415.725,A -85,B 0,C 180,E1 -5505.584,E2 -5505.584} C_VEL
LIN {X 0,Y 510.811,Z 388.959,A -85,B 0,C 180,E1 -5508.864,E2 -5508.864} C_VEL
LIN {X 0,Y 511.251,Z 365.446,A -85,B 0,C 180,E1 -5511.787,E2 -5511.787} C_VEL
LIN {X 0,Y 511.756,Z 343.985,A -85,B 0,C 180,E1 -5514.51,E2 -5514.51} C_VEL
LIN {X 0,Y 512.019,Z 329.149,A -85,B 0,C 180,E1 -5516.443,E2 -5516.443} C_VEL
LIN {X 0,Y 509.851,Z 317.979,A -85,B 0,C 180,E1 -5518.043,E2 -5518.043} C_VEL
LIN {X 0,Y 509.848,Z 317.982,A -85,B 0,C 180,E1 -5520.666,E2 -5520.666} C_VEL
LIN {X 0,Y 509.845,Z 317.976,A -85,B 0,C 180,E1 -5523.462,E2 -5523.462} C_VEL
LIN {X 0,Y 509.812,Z 317.983,A -85,B 0,C 180,E1 -5526.354,E2 -5526.354} C_VEL
LIN {X 0,Y 509.835,Z 317.976,A -85,B 0,C 180,E1 -5529.354,E2 -5529.354} C_VEL
LIN {X 0,Y 509.805,Z 317.984,A -85,B 0,C 180,E1 -5532.493,E2 -5532.493} C_VEL
LIN {X 0,Y 509.842,Z 317.974,A -85,B 0,C 180,E1 -5535.33,E2 -5535.33} C_VEL
LIN {X 0,Y 509.832,Z 317.977,A -85,B 0,C 180,E1 -5538.572,E2 -5538.572} C_VEL
LIN {X 0,Y 509.816,Z 317.982,A -85,B 0,C 180,E1 -5541.792,E2 -5541.792} C_VEL
LIN {X 0,Y 509.81,Z 317.978,A -85,B 0,C 180,E1 -5544.62,E2 -5544.62} C_VEL
LIN {X 0,Y 509.86,Z 317.974,A -85,B 0,C 180,E1 -5547.48,E2 -5547.48} C_VEL
LIN {X 0,Y 509.831,Z 317.978,A -85,B 0,C 180,E1 -5550.28,E2 -5550.28} C_VEL
LIN {X 0,Y 509.815,Z 317.977,A -85,B 0,C 180,E1 -5552.94,E2 -5552.94} C_VEL
LIN {X 0,Y 509.824,Z 317.983,A -85,B 0,C 180,E1 -5555.571,E2 -5555.571} C_VEL
LIN {X 0,Y 509.803,Z 317.982,A -85,B 0,C 180,E1 -5558.147,E2 -5558.147} C_VEL
LIN {X 0,Y 509.827,Z 317.977,A -85,B 0,C 180,E1 -5560.68,E2 -5560.68} C_VEL
LIN {X 0,Y 509.848,Z 317.978,A -85,B 0,C 180,E1 -5563.173,E2 -5563.173} C_VEL
LIN {X 0,Y 509.85,Z 317.981,A -85,B 0,C 180,E1 -5565.633,E2 -5565.633} C_VEL
LIN {X 0,Y 509.854,Z 317.978,A -85,B 0,C 180,E1 -5566.774,E2 -5566.774} C_VEL
LIN {X 0,Y 512.164,Z 325.757,A -85,B 0,C 180,E1 -5566.977,E2 -5566.977} C_VEL
LIN {X 0,Y 511.559,Z 407.946,A -85,B 0,C 180,E1 -5568.233,E2 -5568.233} C_VEL
LIN {X 0,Y 511.476,Z 421.405,A -85,B 0,C 180,E1 -5568.608,E2 -5568.608} C_VEL
LIN {X 0,Y 511.329,Z 433.585,A -85,B 0,C 180,E1 -5569.106,E2 -5569.106} C_VEL
LIN {X 0,Y 511.131,Z 444.496,A -85,B 0,C 180,E1 -5569.703,E2 -5569.703} C_VEL
LIN {X 0,Y 510.836,Z 455.864,A -85,B 0,C 180,E1 -5570.497,E2 -5570.497} C_VEL
LIN {X 0,Y 510.586,Z 466.076,A -85,B 0,C 180,E1 -5571.391,E2 -5571.391} C_VEL
LIN {X 0,Y 510.293,Z 474.99,A -85,B 0,C 180,E1 -5572.352,E2 -5572.352} C_VEL
LIN {X 0,Y 510.025,Z 483.545,A -85,B 0,C 180,E1 -5573.494,E2 -5573.494} C_VEL
LIN {X 0,Y 509.952,Z 490.588,A -85,B 0,C 180,E1 -5574.662,E2 -5574.662} C_VEL
LIN {X 0,Y 509.722,Z 495.474,A -85,B 0,C 180,E1 -5575.651,E2 -5575.651} C_VEL
LIN {X 0,Y 509.541,Z 500.19,A -85,B 0,C 180,E1 -5576.837,E2 -5576.837} C_VEL
LIN {X 0,Y 509.536,Z 503.78,A -85,B 0,C 180,E1 -5578.024,E2 -5578.024} C_VEL
LIN {X 0,Y 509.375,Z 506.386,A -85,B 0,C 180,E1 -5579.209,E2 -5579.209} C_VEL
LIN {X 0,Y 509.361,Z 508.409,A -85,B 0,C 180,E1 -5580.79,E2 -5580.79} C_VEL
LIN {X 0,Y 509.31,Z 508.795,A -85,B 0,C 180,E1 -5582.372,E2 -5582.372} C_VEL
LIN {X 0,Y 509.383,Z 508.405,A -85,B 0,C 180,E1 -5583.163,E2 -5583.163} C_VEL
LIN {X 0,Y 509.389,Z 507.635,A -85,B 0,C 180,E1 -5583.955,E2 -5583.955} C_VEL
LIN {X 0,Y 509.394,Z 506.424,A -85,B 0,C 180,E1 -5584.748,E2 -5584.748} C_VEL
LIN {X 0,Y 509.508,Z 503.848,A -85,B 0,C 180,E1 -5585.938,E2 -5585.938} C_VEL
LIN {X 0,Y 509.566,Z 500.269,A -85,B 0,C 180,E1 -5587.13,E2 -5587.13} C_VEL
LIN {X 0,Y 509.655,Z 495.57,A -85,B 0,C 180,E1 -5588.325,E2 -5588.325} C_VEL
LIN {X 0,Y 509.854,Z 488.483,A -85,B 0,C 180,E1 -5589.721,E2 -5589.721} C_VEL
LIN {X 0,Y 510.054,Z 480.744,A -85,B 0,C 180,E1 -5590.921,E2 -5590.921} C_VEL
LIN {X 0,Y 510.3,Z 471.344,A -85,B 0,C 180,E1 -5592.085,E2 -5592.085} C_VEL
LIN {X 0,Y 510.581,Z 460.866,A -85,B 0,C 180,E1 -5593.127,E2 -5593.127} C_VEL
LIN {X 0,Y 510.857,Z 450.76,A -85,B 0,C 180,E1 -5593.931,E2 -5593.931} C_VEL
LIN {X 0,Y 511.195,Z 439.728,A -85,B 0,C 180,E1 -5594.632,E2 -5594.632} C_VEL
LIN {X 0,Y 511.427,Z 427.819,A -85,B 0,C 180,E1 -5595.222,E2 -5595.222} C_VEL
LIN {X 0,Y 511.569,Z 414.991,A -85,B 0,C 180,E1 -5595.681,E2 -5595.681} C_VEL
LIN {X 0,Y 511.65,Z 402.473,A -85,B 0,C 180,E1 -5595.97,E2 -5595.97} C_VEL
LIN {X 0,Y 512.02,Z 324.695,A -85,B 0,C 180,E1 -5597.127,E2 -5597.127} C_VEL
LIN {X 0,Y 509.88,Z 317.972,A -85,B 0,C 180,E1 -5597.315,E2 -5597.315} C_VEL
LIN {X 0,Y 509.888,Z 317.973,A -85,B 0,C 180,E1 -5600.401,E2 -5600.401} C_VEL
LIN {X 0,Y 509.83,Z 317.974,A -85,B 0,C 180,E1 -5603.563,E2 -5603.563} C_VEL
LIN {X 0,Y 509.912,Z 317.968,A -85,B 0,C 180,E1 -5606.378,E2 -5606.378} C_VEL
LIN {X 0,Y 509.875,Z 317.974,A -85,B 0,C 180,E1 -5608.844,E2 -5608.844} C_VEL
LIN {X 0,Y 509.819,Z 317.975,A -85,B 0,C 180,E1 -5611.59,E2 -5611.59} C_VEL
LIN {X 0,Y 509.838,Z 317.979,A -85,B 0,C 180,E1 -5614.414,E2 -5614.414} C_VEL
LIN {X 0,Y 509.816,Z 317.976,A -85,B 0,C 180,E1 -5617.34,E2 -5617.34} C_VEL
LIN {X 0,Y 509.837,Z 317.979,A -85,B 0,C 180,E1 -5620.382,E2 -5620.382} C_VEL
LIN {X 0,Y 509.852,Z 317.973,A -85,B 0,C 180,E1 -5621.926,E2 -5621.926} C_VEL
LIN {X 0,Y 509.148,Z 318.067,A -85,B 0,C 180,E1 -5622.585,E2 -5622.585} C_VEL
LIN {X 0,Y 506.259,Z 318.423,A -85,B 0,C 180,E1 -5623.654,E2 -5623.654} C_VEL
LIN {X 0,Y 503.854,Z 318.727,A -85,B 0,C 180,E1 -5624.516,E2 -5624.516} C_VEL
LIN {X 0,Y 502.848,Z 318.845,A -85,B 0,C 180,E1 -5625.182,E2 -5625.182} C_VEL
LIN {X 0,Y 502.78,Z 318.853,A -85,B 0,C 180,E1 -5625.407,E2 -5625.407} C_VEL
LIN {X 0,Y 502.793,Z 318.853,A -85,B 0,C 180,E1 -5627.86,E2 -5627.86} C_VEL
LIN {X 0,Y 502.8,Z 318.851,A -85,B 0,C 180,E1 -5631.024,E2 -5631.024} C_VEL
LIN {X 0,Y 502.782,Z 318.857,A -85,B 0,C 180,E1 -5634.167,E2 -5634.167} C_VEL
LIN {X 0,Y 502.831,Z 318.847,A -85,B 0,C 180,E1 -5636.993,E2 -5636.993} C_VEL
LIN {X 0,Y 502.813,Z 318.853,A -85,B 0,C 180,E1 -5640.065,E2 -5640.065} C_VEL
LIN {X 0,Y 502.832,Z 318.851,A -85,B 0,C 180,E1 -5642.533,E2 -5642.533} C_VEL
LIN {X 0,Y 502.827,Z 318.847,A -85,B 0,C 180,E1 -5645.298,E2 -5645.298} C_VEL
LIN {X 0,Y 502.779,Z 318.856,A -85,B 0,C 180,E1 -5647.826,E2 -5647.826} C_VEL
LIN {X 0,Y 502.824,Z 318.853,A -85,B 0,C 180,E1 -5650.4,E2 -5650.4} C_VEL
LIN {X 0,Y 502.831,Z 318.847,A -85,B 0,C 180,E1 -5652.932,E2 -5652.932} C_VEL
LIN {X 0,Y 502.843,Z 318.846,A -85,B 0,C 180,E1 -5655.429,E2 -5655.429} C_VEL
LIN {X 0,Y 502.875,Z 318.842,A -85,B 0,C 180,E1 -5658.717,E2 -5658.717} C_VEL
LIN {X 0,Y 502.899,Z 318.843,A -85,B 0,C 180,E1 -5661.967,E2 -5661.967} C_VEL
LIN {X 0,Y 502.936,Z 318.838,A -85,B 0,C 180,E1 -5664.387,E2 -5664.387} C_VEL
LIN {X 0,Y 503.023,Z 318.825,A -85,B 0,C 180,E1 -5667.598,E2 -5667.598} C_VEL
LIN {X 0,Y 503.026,Z 318.828,A -85,B 0,C 180,E1 -5670,E2 -5670} C_VEL
LIN {X 0,Y 503.023,Z 318.826,A -85,B 0,C 180,E1 -5672.402,E2 -5672.402} C_VEL
LIN {X 0,Y 502.936,Z 318.837,A -85,B 0,C 180,E1 -5675.614,E2 -5675.614} C_VEL
LIN {X 0,Y 502.899,Z 318.845,A -85,B 0,C 180,E1 -5678.034,E2 -5678.034} C_VEL
LIN {X 0,Y 502.876,Z 318.842,A -85,B 0,C 180,E1 -5681.283,E2 -5681.283} C_VEL
LIN {X 0,Y 502.843,Z 318.846,A -85,B 0,C 180,E1 -5684.571,E2 -5684.571} C_VEL
LIN {X 0,Y 502.86,Z 318.85,A -85,B 0,C 180,E1 -5687.907,E2 -5687.907} C_VEL
LIN {X 0,Y 502.827,Z 318.848,A -85,B 0,C 180,E1 -5690.537,E2 -5690.537} C_VEL
LIN {X 0,Y 502.796,Z 318.851,A -85,B 0,C 180,E1 -5693.041,E2 -5693.041} C_VEL
LIN {X 0,Y 502.839,Z 318.851,A -85,B 0,C 180,E1 -5695.676,E2 -5695.676} C_VEL
LIN {X 0,Y 502.839,Z 318.847,A -85,B 0,C 180,E1 -5698.373,E2 -5698.373} C_VEL
LIN {X 0,Y 502.793,Z 318.856,A -85,B 0,C 180,E1 -5701.5,E2 -5701.5} C_VEL
LIN {X 0,Y 502.805,Z 318.85,A -85,B 0,C 180,E1 -5704.445,E2 -5704.445} C_VEL
LIN {X 0,Y 502.78,Z 318.855,A -85,B 0,C 180,E1 -5707.179,E2 -5707.179} C_VEL
LIN {X 0,Y 502.788,Z 318.856,A -85,B 0,C 180,E1 -5710.016,E2 -5710.016} C_VEL
LIN {X 0,Y 502.803,Z 318.852,A -85,B 0,C 180,E1 -5712.2,E2 -5712.2} C_VEL
LIN {X 0,Y 502.786,Z 318.857,A -85,B 0,C 180,E1 -5715.471,E2 -5715.471} C_VEL
LIN {X 0,Y 502.82,Z 318.849,A -85,B 0,C 180,E1 -5718.935,E2 -5718.935} C_VEL
LIN {X 0,Y 502.794,Z 318.853,A -85,B 0,C 180,E1 -5722.047,E2 -5722.047} C_VEL
LIN {X 0,Y 502.797,Z 318.854,A -85,B 0,C 180,E1 -5725.035,E2 -5725.035} C_VEL
LIN {X 0,Y 502.784,Z 318.855,A -85,B 0,C 180,E1 -5727.916,E2 -5727.916} C_VEL
LIN {X 0,Y 502.825,Z 318.848,A -85,B 0,C 180,E1 -5730.713,E2 -5730.713} C_VEL
LIN {X 0,Y 502.866,Z 318.849,A -85,B 0,C 180,E1 -5733.44,E2 -5733.44} C_VEL
LIN {X 0,Y 502.826,Z 318.93,A -85,B 0,C 180,E1 -5736.585,E2 -5736.585} C_VEL
LIN {X 0,Y 505.307,Z 326.893,A -85,B 0,C 180,E1 -5736.788,E2 -5736.788} C_VEL
LIN {X 0,Y 504.774,Z 406.615,A -85,B 0,C 180,E1 -5738,E2 -5738} C_VEL
LIN {X 0,Y 504.591,Z 419.385,A -85,B 0,C 180,E1 -5738.341,E2 -5738.341} C_VEL
LIN {X 0,Y 504.447,Z 431.486,A -85,B 0,C 180,E1 -5738.824,E2 -5738.824} C_VEL
LIN {X 0,Y 504.205,Z 443.383,A -85,B 0,C 180,E1 -5739.462,E2 -5739.462} C_VEL
LIN {X 0,Y 503.888,Z 454.585,A -85,B 0,C 180,E1 -5740.231,E2 -5740.231} C_VEL
LIN {X 0,Y 503.587,Z 465.375,A -85,B 0,C 180,E1 -5741.172,E2 -5741.172} C_VEL
LIN {X 0,Y 503.311,Z 474.147,A -85,B 0,C 180,E1 -5742.11,E2 -5742.11} C_VEL
LIN {X 0,Y 503.042,Z 482.169,A -85,B 0,C 180,E1 -5743.149,E2 -5743.149} C_VEL
LIN {X 0,Y 502.817,Z 489.943,A -85,B 0,C 180,E1 -5744.392,E2 -5744.392} C_VEL
LIN {X 0,Y 502.669,Z 495.189,A -85,B 0,C 180,E1 -5745.424,E2 -5745.424} C_VEL
LIN {X 0,Y 502.488,Z 500.219,A -85,B 0,C 180,E1 -5746.658,E2 -5746.658} C_VEL
LIN {X 0,Y 502.453,Z 504.063,A -85,B 0,C 180,E1 -5747.889,E2 -5747.889} C_VEL
LIN {X 0,Y 502.387,Z 506.032,A -85,B 0,C 180,E1 -5748.706,E2 -5748.706} C_VEL
LIN {X 0,Y 502.323,Z 507.578,A -85,B 0,C 180,E1 -5749.521,E2 -5749.521} C_VEL
LIN {X 0,Y 502.318,Z 508.657,A -85,B 0,C 180,E1 -5750.335,E2 -5750.335} C_VEL
LIN {X 0,Y 502.329,Z 509.628,A -85,B 0,C 180,E1 -5751.958,E2 -5751.958} C_VEL
LIN {X 0,Y 502.411,Z 509.183,A -85,B 0,C 180,E1 -5753.313,E2 -5753.313} C_VEL
LIN {X 0,Y 502.401,Z 508.02,A -85,B 0,C 180,E1 -5754.381,E2 -5754.381} C_VEL
LIN {X 0,Y 502.468,Z 506.683,A -85,B 0,C 180,E1 -5755.186,E2 -5755.186} C_VEL
LIN {X 0,Y 502.491,Z 503.874,A -85,B 0,C 180,E1 -5756.392,E2 -5756.392} C_VEL
LIN {X 0,Y 502.577,Z 500.03,A -85,B 0,C 180,E1 -5757.596,E2 -5757.596} C_VEL
LIN {X 0,Y 502.678,Z 495.046,A -85,B 0,C 180,E1 -5758.799,E2 -5758.799} C_VEL
LIN {X 0,Y 502.979,Z 487.571,A -85,B 0,C 180,E1 -5760.201,E2 -5760.201} C_VEL
LIN {X 0,Y 503.158,Z 480.941,A -85,B 0,C 180,E1 -5761.201,E2 -5761.201} C_VEL
LIN {X 0,Y 503.453,Z 472.934,A -85,B 0,C 180,E1 -5762.2,E2 -5762.2} C_VEL
LIN {X 0,Y 503.757,Z 463.086,A -85,B 0,C 180,E1 -5763.199,E2 -5763.199} C_VEL
LIN {X 0,Y 504.03,Z 452.092,A -85,B 0,C 180,E1 -5764.098,E2 -5764.098} C_VEL
LIN {X 0,Y 504.31,Z 441.255,A -85,B 0,C 180,E1 -5764.797,E2 -5764.797} C_VEL
LIN {X 0,Y 504.508,Z 427.991,A -85,B 0,C 180,E1 -5765.446,E2 -5765.446} C_VEL
LIN {X 0,Y 504.671,Z 415.849,A -85,B 0,C 180,E1 -5765.87,E2 -5765.87} C_VEL
LIN {X 0,Y 504.739,Z 402.079,A -85,B 0,C 180,E1 -5766.17,E2 -5766.17} C_VEL
LIN {X 0,Y 505.358,Z 326.926,A -85,B 0,C 180,E1 -5767.312,E2 -5767.312} C_VEL
LIN {X 0,Y 502.868,Z 318.852,A -85,B 0,C 180,E1 -5767.522,E2 -5767.522} C_VEL
LIN {X 0,Y 502.771,Z 318.863,A -85,B 0,C 180,E1 -5770.47,E2 -5770.47} C_VEL
LIN {X 0,Y 502.805,Z 318.854,A -85,B 0,C 180,E1 -5772.923,E2 -5772.923} C_VEL
LIN {X 0,Y 502.852,Z 318.846,A -85,B 0,C 180,E1 -5775.4,E2 -5775.4} C_VEL
LIN {X 0,Y 502.793,Z 318.858,A -85,B 0,C 180,E1 -5778.102,E2 -5778.102} C_VEL
LIN {X 0,Y 502.759,Z 318.858,A -85,B 0,C 180,E1 -5781.313,E2 -5781.313} C_VEL
LIN {X 0,Y 502.76,Z 318.859,A -85,B 0,C 180,E1 -5783.916,E2 -5783.916} C_VEL
LIN {X 0,Y 502.761,Z 318.86,A -85,B 0,C 180,E1 -5786.572,E2 -5786.572} C_VEL
LIN {X 0,Y 502.795,Z 318.851,A -85,B 0,C 180,E1 -5789.29,E2 -5789.29} C_VEL
LIN {X 0,Y 502.782,Z 318.859,A -85,B 0,C 180,E1 -5792.085,E2 -5792.085} C_VEL
LIN {X 0,Y 502.787,Z 318.85,A -85,B 0,C 180,E1 -5794.967,E2 -5794.967} C_VEL
LIN {X 0,Y 502.767,Z 318.855,A -85,B 0,C 180,E1 -5798.481,E2 -5798.481} C_VEL
LIN {X 0,Y 502.767,Z 318.853,A -85,B 0,C 180,E1 -5801.072,E2 -5801.072} C_VEL
LIN {X 0,Y 502.79,Z 318.852,A -85,B 0,C 180,E1 -5804.53,E2 -5804.53} C_VEL
LIN {X 0,Y 502.799,Z 318.858,A -85,B 0,C 180,E1 -5807.86,E2 -5807.86} C_VEL
LIN {X 0,Y 502.797,Z 318.852,A -85,B 0,C 180,E1 -5811.023,E2 -5811.023} C_VEL
LIN {X 0,Y 502.773,Z 318.856,A -85,B 0,C 180,E1 -5814.17,E2 -5814.17} C_VEL
LIN {X 0,Y 502.835,Z 318.848,A -85,B 0,C 180,E1 -5816.994,E2 -5816.994} C_VEL
LIN {X 0,Y 502.819,Z 318.853,A -85,B 0,C 180,E1 -5820.065,E2 -5820.065} C_VEL
LIN {X 0,Y 502.851,Z 318.874,A -85,B 0,C 180,E1 -5821.315,E2 -5821.315} C_VEL
LIN {X 0,Y 505.678,Z 331.988,A -85,B 0,C 180,E1 -5823.229,E2 -5823.229} C_VEL
LIN {X 0,Y 505.334,Z 346.555,A -85,B 0,C 180,E1 -5825.16,E2 -5825.16} C_VEL
LIN {X 0,Y 504.54,Z 372.613,A -85,B 0,C 180,E1 -5828.552,E2 -5828.552} C_VEL
LIN {X 0,Y 503.818,Z 400.637,A -85,B 0,C 180,E1 -5832.128,E2 -5832.128} C_VEL
LIN {X 0,Y 503.403,Z 416.859,A -85,B 0,C 180,E1 -5834.185,E2 -5834.185} C_VEL
LIN {X 0,Y 505.253,Z 433.937,A -85,B 0,C 180,E1 -5834.522,E2 -5834.522} C_VEL
LIN {X 0,Y 504.616,Z 525.363,A -85,B 0,C 180,E1 -5835.893,E2 -5835.893} C_VEL
LIN {X 0,Y 504.342,Z 538.397,A -85,B 0,C 180,E1 -5836.219,E2 -5836.219} C_VEL
LIN {X 0,Y 504.043,Z 551,A -85,B 0,C 180,E1 -5836.699,E2 -5836.699} C_VEL
LIN {X 0,Y 503.705,Z 562.796,A -85,B 0,C 180,E1 -5837.305,E2 -5837.305} C_VEL
LIN {X 0,Y 503.411,Z 573.607,A -85,B 0,C 180,E1 -5838.014,E2 -5838.014} C_VEL
LIN {X 0,Y 503.052,Z 584.655,A -85,B 0,C 180,E1 -5838.925,E2 -5838.925} C_VEL
LIN {X 0,Y 502.769,Z 594.586,A -85,B 0,C 180,E1 -5839.937,E2 -5839.937} C_VEL
LIN {X 0,Y 502.572,Z 602.738,A -85,B 0,C 180,E1 -5840.948,E2 -5840.948} C_VEL
LIN {X 0,Y 502.393,Z 610.726,A -85,B 0,C 180,E1 -5842.161,E2 -5842.161} C_VEL
LIN {X 0,Y 502.278,Z 617.431,A -85,B 0,C 180,E1 -5843.441,E2 -5843.441} C_VEL
LIN {X 0,Y 502.202,Z 622.909,A -85,B 0,C 180,E1 -5844.781,E2 -5844.781} C_VEL
LIN {X 0,Y 502.248,Z 626.64,A -85,B 0,C 180,E1 -5845.988,E2 -5845.988} C_VEL
LIN {X 0,Y 502.229,Z 628.555,A -85,B 0,C 180,E1 -5846.791,E2 -5846.791} C_VEL
LIN {X 0,Y 502.168,Z 629.987,A -85,B 0,C 180,E1 -5847.594,E2 -5847.594} C_VEL
LIN {X 0,Y 502.129,Z 631.001,A -85,B 0,C 180,E1 -5848.396,E2 -5848.396} C_VEL
LIN {X 0,Y 502.12,Z 631.608,A -85,B 0,C 180,E1 -5849.198,E2 -5849.198} C_VEL
LIN {X 0,Y 502.126,Z 631.812,A -85,B 0,C 180,E1 -5850,E2 -5850} C_VEL
LIN {X 0,Y 502.124,Z 631.57,A -85,B 0,C 180,E1 -5850.802,E2 -5850.802} C_VEL
LIN {X 0,Y 502.138,Z 630.924,A -85,B 0,C 180,E1 -5851.604,E2 -5851.604} C_VEL
LIN {X 0,Y 502.18,Z 629.864,A -85,B 0,C 180,E1 -5852.406,E2 -5852.406} C_VEL
LIN {X 0,Y 502.232,Z 628.386,A -85,B 0,C 180,E1 -5853.209,E2 -5853.209} C_VEL
LIN {X 0,Y 502.239,Z 625.293,A -85,B 0,C 180,E1 -5854.414,E2 -5854.414} C_VEL
LIN {X 0,Y 502.284,Z 621.115,A -85,B 0,C 180,E1 -5855.621,E2 -5855.621} C_VEL
LIN {X 0,Y 502.337,Z 614.799,A -85,B 0,C 180,E1 -5857.011,E2 -5857.011} C_VEL
LIN {X 0,Y 502.478,Z 607.678,A -85,B 0,C 180,E1 -5858.242,E2 -5858.242} C_VEL
LIN {X 0,Y 502.637,Z 598.958,A -85,B 0,C 180,E1 -5859.456,E2 -5859.456} C_VEL
LIN {X 0,Y 502.871,Z 588.976,A -85,B 0,C 180,E1 -5860.57,E2 -5860.57} C_VEL
LIN {X 0,Y 503.201,Z 578.949,A -85,B 0,C 180,E1 -5861.48,E2 -5861.48} C_VEL
LIN {X 0,Y 503.43,Z 568.263,A -85,B 0,C 180,E1 -5862.271,E2 -5862.271} C_VEL
LIN {X 0,Y 503.716,Z 556.683,A -85,B 0,C 180,E1 -5862.95,E2 -5862.95} C_VEL
LIN {X 0,Y 504.089,Z 544.24,A -85,B 0,C 180,E1 -5863.505,E2 -5863.505} C_VEL
LIN {X 0,Y 504.366,Z 530.688,A -85,B 0,C 180,E1 -5863.934,E2 -5863.934} C_VEL
LIN {X 0,Y 504.642,Z 515.68,A -85,B 0,C 180,E1 -5864.209,E2 -5864.209} C_VEL
LIN {X 0,Y 505.066,Z 431.419,A -85,B 0,C 180,E1 -5865.484,E2 -5865.484} C_VEL
LIN {X 0,Y 503.252,Z 414.474,A -85,B 0,C 180,E1 -5865.826,E2 -5865.826} C_VEL
LIN {X 0,Y 503.77,Z 389.589,A -85,B 0,C 180,E1 -5868.927,E2 -5868.927} C_VEL
LIN {X 0,Y 504.261,Z 366.197,A -85,B 0,C 180,E1 -5871.89,E2 -5871.89} C_VEL
LIN {X 0,Y 504.823,Z 344.577,A -85,B 0,C 180,E1 -5874.686,E2 -5874.686} C_VEL
LIN {X 0,Y 505.077,Z 330.039,A -85,B 0,C 180,E1 -5876.62,E2 -5876.62} C_VEL
LIN {X 0,Y 502.798,Z 318.858,A -85,B 0,C 180,E1 -5878.285,E2 -5878.285} C_VEL
LIN {X 0,Y 502.799,Z 318.856,A -85,B 0,C 180,E1 -5881.143,E2 -5881.143} C_VEL
LIN {X 0,Y 502.792,Z 318.857,A -85,B 0,C 180,E1 -5883.995,E2 -5883.995} C_VEL
LIN {X 0,Y 502.767,Z 318.856,A -85,B 0,C 180,E1 -5887.176,E2 -5887.176} C_VEL
LIN {X 0,Y 502.773,Z 318.861,A -85,B 0,C 180,E1 -5890.017,E2 -5890.017} C_VEL
LIN {X 0,Y 502.773,Z 318.862,A -85,B 0,C 180,E1 -5892.195,E2 -5892.195} C_VEL
LIN {X 0,Y 502.788,Z 318.854,A -85,B 0,C 180,E1 -5895.47,E2 -5895.47} C_VEL
LIN {X 0,Y 502.773,Z 318.854,A -85,B 0,C 180,E1 -5898.929,E2 -5898.929} C_VEL
LIN {X 0,Y 502.762,Z 318.861,A -85,B 0,C 180,E1 -5902.043,E2 -5902.043} C_VEL
LIN {X 0,Y 502.785,Z 318.852,A -85,B 0,C 180,E1 -5905.033,E2 -5905.033} C_VEL
LIN {X 0,Y 502.78,Z 318.859,A -85,B 0,C 180,E1 -5907.915,E2 -5907.915} C_VEL
LIN {X 0,Y 502.793,Z 318.852,A -85,B 0,C 180,E1 -5910.71,E2 -5910.71} C_VEL
LIN {X 0,Y 502.772,Z 318.859,A -85,B 0,C 180,E1 -5913.461,E2 -5913.461} C_VEL
LIN {X 0,Y 502.758,Z 318.861,A -85,B 0,C 180,E1 -5916.084,E2 -5916.084} C_VEL
LIN {X 0,Y 502.76,Z 318.858,A -85,B 0,C 180,E1 -5918.687,E2 -5918.687} C_VEL
LIN {X 0,Y 502.795,Z 318.856,A -85,B 0,C 180,E1 -5921.897,E2 -5921.897} C_VEL
LIN {X 0,Y 502.838,Z 318.85,A -85,B 0,C 180,E1 -5924.665,E2 -5924.665} C_VEL
LIN {X 0,Y 502.828,Z 318.986,A -85,B 0,C 180,E1 -5926.562,E2 -5926.562} C_VEL
LIN {X 0,Y 505.331,Z 327.038,A -85,B 0,C 180,E1 -5926.779,E2 -5926.779} C_VEL
LIN {X 0,Y 504.652,Z 409.195,A -85,B 0,C 180,E1 -5928.069,E2 -5928.069} C_VEL
LIN {X 0,Y 504.583,Z 422.528,A -85,B 0,C 180,E1 -5928.45,E2 -5928.45} C_VEL
LIN {X 0,Y 504.426,Z 434.647,A -85,B 0,C 180,E1 -5928.955,E2 -5928.955} C_VEL
LIN {X 0,Y 504.215,Z 445.528,A -85,B 0,C 180,E1 -5929.56,E2 -5929.56} C_VEL
LIN {X 0,Y 503.906,Z 456.878,A -85,B 0,C 180,E1 -5930.365,E2 -5930.365} C_VEL
LIN {X 0,Y 503.646,Z 467.076,A -85,B 0,C 180,E1 -5931.271,E2 -5931.271} C_VEL
LIN {X 0,Y 503.329,Z 475.977,A -85,B 0,C 180,E1 -5932.245,E2 -5932.245} C_VEL
LIN {X 0,Y 503.046,Z 484.528,A -85,B 0,C 180,E1 -5933.403,E2 -5933.403} C_VEL
LIN {X 0,Y 502.967,Z 491.562,A -85,B 0,C 180,E1 -5934.588,E2 -5934.588} C_VEL
LIN {X 0,Y 502.715,Z 496.439,A -85,B 0,C 180,E1 -5935.59,E2 -5935.59} C_VEL
LIN {X 0,Y 502.517,Z 501.145,A -85,B 0,C 180,E1 -5936.793,E2 -5936.793} C_VEL
LIN {X 0,Y 502.513,Z 504.719,A -85,B 0,C 180,E1 -5937.996,E2 -5937.996} C_VEL
LIN {X 0,Y 502.35,Z 507.306,A -85,B 0,C 180,E1 -5939.198,E2 -5939.198} C_VEL
LIN {X 0,Y 502.328,Z 508.503,A -85,B 0,C 180,E1 -5940,E2 -5940} C_VEL
LIN {X 0,Y 502.335,Z 509.298,A -85,B 0,C 180,E1 -5940.801,E2 -5940.801} C_VEL
LIN {X 0,Y 502.265,Z 509.652,A -85,B 0,C 180,E1 -5942.405,E2 -5942.405} C_VEL
LIN {X 0,Y 502.336,Z 509.24,A -85,B 0,C 180,E1 -5943.208,E2 -5943.208} C_VEL
LIN {X 0,Y 502.351,Z 508.44,A -85,B 0,C 180,E1 -5944.011,E2 -5944.011} C_VEL
LIN {X 0,Y 502.357,Z 507.205,A -85,B 0,C 180,E1 -5944.815,E2 -5944.815} C_VEL
LIN {X 0,Y 502.489,Z 504.581,A -85,B 0,C 180,E1 -5946.021,E2 -5946.021} C_VEL
LIN {X 0,Y 502.565,Z 500.95,A -85,B 0,C 180,E1 -5947.23,E2 -5947.23} C_VEL
LIN {X 0,Y 502.662,Z 496.195,A -85,B 0,C 180,E1 -5948.441,E2 -5948.441} C_VEL
LIN {X 0,Y 502.839,Z 490.163,A -85,B 0,C 180,E1 -5949.655,E2 -5949.655} C_VEL
LIN {X 0,Y 503.069,Z 482.63,A -85,B 0,C 180,E1 -5950.871,E2 -5950.871} C_VEL
LIN {X 0,Y 503.267,Z 475.015,A -85,B 0,C 180,E1 -5951.874,E2 -5951.874} C_VEL
LIN {X 0,Y 503.55,Z 465.468,A -85,B 0,C 180,E1 -5952.903,E2 -5952.903} C_VEL
LIN {X 0,Y 503.882,Z 454.929,A -85,B 0,C 180,E1 -5953.819,E2 -5953.819} C_VEL
LIN {X 0,Y 504.185,Z 443.162,A -85,B 0,C 180,E1 -5954.634,E2 -5954.634} C_VEL
LIN {X 0,Y 504.462,Z 430.541,A -85,B 0,C 180,E1 -5955.297,E2 -5955.297} C_VEL
LIN {X 0,Y 504.656,Z 417.291,A -85,B 0,C 180,E1 -5955.805,E2 -5955.805} C_VEL
LIN {X 0,Y 504.763,Z 405.043,A -85,B 0,C 180,E1 -5956.113,E2 -5956.113} C_VEL
LIN {X 0,Y 505.186,Z 326.235,A -85,B 0,C 180,E1 -5957.315,E2 -5957.315} C_VEL
LIN {X 0,Y 502.861,Z 318.846,A -85,B 0,C 180,E1 -5957.513,E2 -5957.513} C_VEL
LIN {X 0,Y 502.831,Z 318.853,A -85,B 0,C 180,E1 -5960.536,E2 -5960.536} C_VEL
LIN {X 0,Y 502.792,Z 318.854,A -85,B 0,C 180,E1 -5963.04,E2 -5963.04} C_VEL
LIN {X 0,Y 502.841,Z 318.845,A -85,B 0,C 180,E1 -5965.675,E2 -5965.675} C_VEL
LIN {X 0,Y 502.84,Z 318.849,A -85,B 0,C 180,E1 -5968.372,E2 -5968.372} C_VEL
LIN {X 0,Y 502.792,Z 318.851,A -85,B 0,C 180,E1 -5971.498,E2 -5971.498} C_VEL
LIN {X 0,Y 502.789,Z 318.853,A -85,B 0,C 180,E1 -5973.995,E2 -5973.995} C_VEL
LIN {X 0,Y 502.777,Z 318.854,A -85,B 0,C 180,E1 -5977.177,E2 -5977.177} C_VEL
LIN {X 0,Y 502.787,Z 318.854,A -85,B 0,C 180,E1 -5980.015,E2 -5980.015} C_VEL
LIN {X 0,Y 502.802,Z 318.854,A -85,B 0,C 180,E1 -5982.199,E2 -5982.199} C_VEL
LIN {X 0,Y 502.78,Z 318.853,A -85,B 0,C 180,E1 -5985.407,E2 -5985.407} C_VEL
LIN {X 0,Y 502.146,Z 318.935,A -85,B 0,C 180,E1 -5986.076,E2 -5986.076} C_VEL
LIN {X 0,Y 499.295,Z 319.292,A -85,B 0,C 180,E1 -5987.161,E2 -5987.161} C_VEL
LIN {X 0,Y 496.869,Z 319.595,A -85,B 0,C 180,E1 -5988.036,E2 -5988.036} C_VEL
LIN {X 0,Y 495.832,Z 319.723,A -85,B 0,C 180,E1 -5988.712,E2 -5988.712} C_VEL
LIN {X 0,Y 495.751,Z 319.73,A -85,B 0,C 180,E1 -5988.94,E2 -5988.94} C_VEL
LIN {X 0,Y 495.749,Z 319.728,A -85,B 0,C 180,E1 -5991.408,E2 -5991.408} C_VEL
LIN {X 0,Y 495.754,Z 319.735,A -85,B 0,C 180,E1 -5994.463,E2 -5994.463} C_VEL
LIN {X 0,Y 495.766,Z 319.726,A -85,B 0,C 180,E1 -5997.405,E2 -5997.405} C_VEL
LIN {X 0,Y 495.764,Z 319.733,A -85,B 0,C 180,E1 -6000.253,E2 -6000.253} C_VEL
LIN {X 0,Y 495.821,Z 319.72,A -85,B 0,C 180,E1 -6003.251,E2 -6003.251} C_VEL
LIN {X 0,Y 495.75,Z 319.73,A -85,B 0,C 180,E1 -6005.725,E2 -6005.725} C_VEL
LIN {X 0,Y 495.741,Z 319.736,A -85,B 0,C 180,E1 -6008.371,E2 -6008.371} C_VEL
LIN {X 0,Y 495.782,Z 319.725,A -85,B 0,C 180,E1 -6010.972,E2 -6010.972} C_VEL
LIN {X 0,Y 495.777,Z 319.726,A -85,B 0,C 180,E1 -6013.53,E2 -6013.53} C_VEL
LIN {X 0,Y 495.792,Z 319.729,A -85,B 0,C 180,E1 -6016.056,E2 -6016.056} C_VEL
LIN {X 0,Y 495.849,Z 319.719,A -85,B 0,C 180,E1 -6018.555,E2 -6018.555} C_VEL
LIN {X 0,Y 495.87,Z 319.718,A -85,B 0,C 180,E1 -6021.852,E2 -6021.852} C_VEL
LIN {X 0,Y 495.893,Z 319.716,A -85,B 0,C 180,E1 -6024.307,E2 -6024.307} C_VEL
LIN {X 0,Y 495.992,Z 319.701,A -85,B 0,C 180,E1 -6027.564,E2 -6027.564} C_VEL
LIN {X 0,Y 495.997,Z 319.704,A -85,B 0,C 180,E1 -6030,E2 -6030} C_VEL
LIN {X 0,Y 495.992,Z 319.701,A -85,B 0,C 180,E1 -6032.436,E2 -6032.436} C_VEL
LIN {X 0,Y 495.893,Z 319.715,A -85,B 0,C 180,E1 -6035.694,E2 -6035.694} C_VEL
LIN {X 0,Y 495.871,Z 319.719,A -85,B 0,C 180,E1 -6038.148,E2 -6038.148} C_VEL
LIN {X 0,Y 495.85,Z 319.719,A -85,B 0,C 180,E1 -6041.445,E2 -6041.445} C_VEL
LIN {X 0,Y 495.788,Z 319.724,A -85,B 0,C 180,E1 -6044.783,E2 -6044.783} C_VEL
LIN {X 0,Y 495.785,Z 319.726,A -85,B 0,C 180,E1 -6047.319,E2 -6047.319} C_VEL
LIN {X 0,Y 495.771,Z 319.733,A -85,B 0,C 180,E1 -6049.891,E2 -6049.891} C_VEL
LIN {X 0,Y 495.764,Z 319.727,A -85,B 0,C 180,E1 -6052.863,E2 -6052.863} C_VEL
LIN {X 0,Y 495.79,Z 319.728,A -85,B 0,C 180,E1 -6056.068,E2 -6056.068} C_VEL
LIN {X 0,Y 495.771,Z 319.726,A -85,B 0,C 180,E1 -6058.815,E2 -6058.815} C_VEL
LIN {X 0,Y 495.756,Z 319.734,A -85,B 0,C 180,E1 -6061.726,E2 -6061.726} C_VEL
LIN {X 0,Y 495.775,Z 319.726,A -85,B 0,C 180,E1 -6064.696,E2 -6064.696} C_VEL
LIN {X 0,Y 495.731,Z 319.736,A -85,B 0,C 180,E1 -6067.562,E2 -6067.562} C_VEL
LIN {X 0,Y 495.766,Z 319.727,A -85,B 0,C 180,E1 -6070.7,E2 -6070.7} C_VEL
LIN {X 0,Y 495.728,Z 319.735,A -85,B 0,C 180,E1 -6074.002,E2 -6074.002} C_VEL
LIN {X 0,Y 495.726,Z 319.735,A -85,B 0,C 180,E1 -6077.118,E2 -6077.118} C_VEL
LIN {X 0,Y 495.759,Z 319.731,A -85,B 0,C 180,E1 -6079.954,E2 -6079.954} C_VEL
LIN {X 0,Y 495.729,Z 319.732,A -85,B 0,C 180,E1 -6082.554,E2 -6082.554} C_VEL
LIN {X 0,Y 495.772,Z 319.732,A -85,B 0,C 180,E1 -6085.457,E2 -6085.457} C_VEL
LIN {X 0,Y 495.756,Z 319.728,A -85,B 0,C 180,E1 -6088.364,E2 -6088.364} C_VEL
LIN {X 0,Y 495.789,Z 319.73,A -85,B 0,C 180,E1 -6091.508,E2 -6091.508} C_VEL
LIN {X 0,Y 495.793,Z 319.725,A -85,B 0,C 180,E1 -6093.933,E2 -6093.933} C_VEL
LIN {X 0,Y 495.786,Z 319.726,A -85,B 0,C 180,E1 -6096.357,E2 -6096.357} C_VEL
LIN {X 0,Y 498.416,Z 327.813,A -85,B 0,C 180,E1 -6096.585,E2 -6096.585} C_VEL
LIN {X 0,Y 497.885,Z 407.133,A -85,B 0,C 180,E1 -6097.816,E2 -6097.816} C_VEL
LIN {X 0,Y 497.729,Z 420.81,A -85,B 0,C 180,E1 -6098.19,E2 -6098.19} C_VEL
LIN {X 0,Y 497.512,Z 433.759,A -85,B 0,C 180,E1 -6098.731,E2 -6098.731} C_VEL
LIN {X 0,Y 497.266,Z 445.986,A -85,B 0,C 180,E1 -6099.417,E2 -6099.417} C_VEL
LIN {X 0,Y 496.925,Z 457.58,A -85,B 0,C 180,E1 -6100.266,E2 -6100.266} C_VEL
LIN {X 0,Y 496.58,Z 467.502,A -85,B 0,C 180,E1 -6101.17,E2 -6101.17} C_VEL
LIN {X 0,Y 496.261,Z 477.29,A -85,B 0,C 180,E1 -6102.274,E2 -6102.274} C_VEL
LIN {X 0,Y 495.971,Z 486.247,A -85,B 0,C 180,E1 -6103.537,E2 -6103.537} C_VEL
LIN {X 0,Y 495.771,Z 492.212,A -85,B 0,C 180,E1 -6104.573,E2 -6104.573} C_VEL
LIN {X 0,Y 495.616,Z 497.251,A -85,B 0,C 180,E1 -6105.632,E2 -6105.632} C_VEL
LIN {X 0,Y 495.446,Z 502.028,A -85,B 0,C 180,E1 -6106.882,E2 -6106.882} C_VEL
LIN {X 0,Y 495.418,Z 505.795,A -85,B 0,C 180,E1 -6108.193,E2 -6108.193} C_VEL
LIN {X 0,Y 495.304,Z 508.2,A -85,B 0,C 180,E1 -6109.371,E2 -6109.371} C_VEL
LIN {X 0,Y 495.27,Z 509.374,A -85,B 0,C 180,E1 -6110.196,E2 -6110.196} C_VEL
LIN {X 0,Y 495.296,Z 510.448,A -85,B 0,C 180,E1 -6111.843,E2 -6111.843} C_VEL
LIN {X 0,Y 495.38,Z 510.081,A -85,B 0,C 180,E1 -6113.268,E2 -6113.268} C_VEL
LIN {X 0,Y 495.36,Z 509.023,A -85,B 0,C 180,E1 -6114.301,E2 -6114.301} C_VEL
LIN {X 0,Y 495.429,Z 507.747,A -85,B 0,C 180,E1 -6115.118,E2 -6115.118} C_VEL
LIN {X 0,Y 495.458,Z 505.022,A -85,B 0,C 180,E1 -6116.341,E2 -6116.341} C_VEL
LIN {X 0,Y 495.559,Z 501.278,A -85,B 0,C 180,E1 -6117.562,E2 -6117.562} C_VEL
LIN {X 0,Y 495.689,Z 496.405,A -85,B 0,C 180,E1 -6118.782,E2 -6118.782} C_VEL
LIN {X 0,Y 495.946,Z 490.215,A -85,B 0,C 180,E1 -6120,E2 -6120} C_VEL
LIN {X 0,Y 496.171,Z 482.533,A -85,B 0,C 180,E1 -6121.218,E2 -6121.218} C_VEL
LIN {X 0,Y 496.49,Z 474.67,A -85,B 0,C 180,E1 -6122.231,E2 -6122.231} C_VEL
LIN {X 0,Y 496.757,Z 465.073,A -85,B 0,C 180,E1 -6123.245,E2 -6123.245} C_VEL
LIN {X 0,Y 497.035,Z 454.292,A -85,B 0,C 180,E1 -6124.156,E2 -6124.156} C_VEL
LIN {X 0,Y 497.364,Z 443.787,A -85,B 0,C 180,E1 -6124.864,E2 -6124.864} C_VEL
LIN {X 0,Y 497.577,Z 432.285,A -85,B 0,C 180,E1 -6125.471,E2 -6125.471} C_VEL
LIN {X 0,Y 497.725,Z 419.041,A -85,B 0,C 180,E1 -6125.978,E2 -6125.978} C_VEL
LIN {X 0,Y 497.831,Z 405.726,A -85,B 0,C 180,E1 -6126.307,E2 -6126.307} C_VEL
LIN {X 0,Y 498.509,Z 327.798,A -85,B 0,C 180,E1 -6127.522,E2 -6127.522} C_VEL
LIN {X 0,Y 495.833,Z 319.722,A -85,B 0,C 180,E1 -6127.763,E2 -6127.763} C_VEL
LIN {X 0,Y 495.816,Z 319.723,A -85,B 0,C 180,E1 -6131.446,E2 -6131.446} C_VEL
LIN {X 0,Y 495.781,Z 319.73,A -85,B 0,C 180,E1 -6134.783,E2 -6134.783} C_VEL
LIN {X 0,Y 495.739,Z 319.733,A -85,B 0,C 180,E1 -6137.321,E2 -6137.321} C_VEL
LIN {X 0,Y 495.709,Z 319.739,A -85,B 0,C 180,E1 -6139.893,E2 -6139.893} C_VEL
LIN {X 0,Y 495.749,Z 319.731,A -85,B 0,C 180,E1 -6142.856,E2 -6142.856} C_VEL
LIN {X 0,Y 495.711,Z 319.741,A -85,B 0,C 180,E1 -6146.073,E2 -6146.073} C_VEL
LIN {X 0,Y 495.723,Z 319.733,A -85,B 0,C 180,E1 -6148.818,E2 -6148.818} C_VEL
LIN {X 0,Y 495.753,Z 319.732,A -85,B 0,C 180,E1 -6151.724,E2 -6151.724} C_VEL
LIN {X 0,Y 495.759,Z 319.727,A -85,B 0,C 180,E1 -6154.691,E2 -6154.691} C_VEL
LIN {X 0,Y 495.704,Z 319.736,A -85,B 0,C 180,E1 -6157.564,E2 -6157.564} C_VEL
LIN {X 0,Y 495.747,Z 319.734,A -85,B 0,C 180,E1 -6160.045,E2 -6160.045} C_VEL
LIN {X 0,Y 495.699,Z 319.733,A -85,B 0,C 180,E1 -6162.886,E2 -6162.886} C_VEL
LIN {X 0,Y 495.727,Z 319.738,A -85,B 0,C 180,E1 -6165.998,E2 -6165.998} C_VEL
LIN {X 0,Y 495.735,Z 319.733,A -85,B 0,C 180,E1 -6169.296,E2 -6169.296} C_VEL
LIN {X 0,Y 495.749,Z 319.734,A -85,B 0,C 180,E1 -6171.408,E2 -6171.408} C_VEL
LIN {X 0,Y 495.747,Z 319.73,A -85,B 0,C 180,E1 -6174.462,E2 -6174.462} C_VEL
LIN {X 0,Y 495.77,Z 319.733,A -85,B 0,C 180,E1 -6177.405,E2 -6177.405} C_VEL
LIN {X 0,Y 495.785,Z 319.728,A -85,B 0,C 180,E1 -6180.721,E2 -6180.721} C_VEL
LIN {X 0,Y 495.809,Z 319.805,A -85,B 0,C 180,E1 -6181.1,E2 -6181.1} C_VEL
LIN {X 0,Y 498.841,Z 334.039,A -85,B 0,C 180,E1 -6183.202,E2 -6183.202} C_VEL
LIN {X 0,Y 498.258,Z 352.196,A -85,B 0,C 180,E1 -6185.633,E2 -6185.633} C_VEL
LIN {X 0,Y 497.476,Z 376.343,A -85,B 0,C 180,E1 -6188.813,E2 -6188.813} C_VEL
LIN {X 0,Y 496.78,Z 401.534,A -85,B 0,C 180,E1 -6192.079,E2 -6192.079} C_VEL
LIN {X 0,Y 496.388,Z 416.201,A -85,B 0,C 180,E1 -6193.966,E2 -6193.966} C_VEL
LIN {X 0,Y 498.384,Z 434.801,A -85,B 0,C 180,E1 -6194.33,E2 -6194.33} C_VEL
LIN {X 0,Y 497.677,Z 526.29,A -85,B 0,C 180,E1 -6195.744,E2 -6195.744} C_VEL
LIN {X 0,Y 497.389,Z 539.361,A -85,B 0,C 180,E1 -6196.101,E2 -6196.101} C_VEL
LIN {X 0,Y 497.046,Z 552.065,A -85,B 0,C 180,E1 -6196.612,E2 -6196.612} C_VEL
LIN {X 0,Y 496.65,Z 563.918,A -85,B 0,C 180,E1 -6197.257,E2 -6197.257} C_VEL
LIN {X 0,Y 496.341,Z 575.224,A -85,B 0,C 180,E1 -6198.048,E2 -6198.048} C_VEL
LIN {X 0,Y 495.987,Z 585.844,A -85,B 0,C 180,E1 -6198.972,E2 -6198.972} C_VEL
LIN {X 0,Y 495.684,Z 595.422,A -85,B 0,C 180,E1 -6199.998,E2 -6199.998} C_VEL
LIN {X 0,Y 495.441,Z 604.665,A -85,B 0,C 180,E1 -6201.228,E2 -6201.228} C_VEL
LIN {X 0,Y 495.305,Z 612.122,A -85,B 0,C 180,E1 -6202.458,E2 -6202.458} C_VEL
LIN {X 0,Y 495.17,Z 618.243,A -85,B 0,C 180,E1 -6203.721,E2 -6203.721} C_VEL
LIN {X 0,Y 495.139,Z 622.048,A -85,B 0,C 180,E1 -6204.706,E2 -6204.706} C_VEL
LIN {X 0,Y 495.182,Z 625.789,A -85,B 0,C 180,E1 -6205.93,E2 -6205.93} C_VEL
LIN {X 0,Y 495.176,Z 627.71,A -85,B 0,C 180,E1 -6206.745,E2 -6206.745} C_VEL
LIN {X 0,Y 495.111,Z 629.145,A -85,B 0,C 180,E1 -6207.559,E2 -6207.559} C_VEL
LIN {X 0,Y 495.076,Z 630.157,A -85,B 0,C 180,E1 -6208.373,E2 -6208.373} C_VEL
LIN {X 0,Y 495.069,Z 630.762,A -85,B 0,C 180,E1 -6209.186,E2 -6209.186} C_VEL
LIN {X 0,Y 495.078,Z 630.962,A -85,B 0,C 180,E1 -6210,E2 -6210} C_VEL
LIN {X 0,Y 495.074,Z 630.714,A -85,B 0,C 180,E1 -6210.813,E2 -6210.813} C_VEL
LIN {X 0,Y 495.087,Z 630.054,A -85,B 0,C 180,E1 -6211.627,E2 -6211.627} C_VEL
LIN {X 0,Y 495.126,Z 628.984,A -85,B 0,C 180,E1 -6212.44,E2 -6212.44} C_VEL
LIN {X 0,Y 495.179,Z 627.493,A -85,B 0,C 180,E1 -6213.254,E2 -6213.254} C_VEL
LIN {X 0,Y 495.181,Z 624.373,A -85,B 0,C 180,E1 -6214.477,E2 -6214.477} C_VEL
LIN {X 0,Y 495.228,Z 620.164,A -85,B 0,C 180,E1 -6215.701,E2 -6215.701} C_VEL
LIN {X 0,Y 495.273,Z 613.797,A -85,B 0,C 180,E1 -6217.112,E2 -6217.112} C_VEL
LIN {X 0,Y 495.42,Z 606.631,A -85,B 0,C 180,E1 -6218.361,E2 -6218.361} C_VEL
LIN {X 0,Y 495.579,Z 597.851,A -85,B 0,C 180,E1 -6219.592,E2 -6219.592} C_VEL
LIN {X 0,Y 495.876,Z 587.807,A -85,B 0,C 180,E1 -6220.72,E2 -6220.72} C_VEL
LIN {X 0,Y 496.186,Z 577.764,A -85,B 0,C 180,E1 -6221.64,E2 -6221.64} C_VEL
LIN {X 0,Y 496.449,Z 566.938,A -85,B 0,C 180,E1 -6222.447,E2 -6222.447} C_VEL
LIN {X 0,Y 496.836,Z 554.214,A -85,B 0,C 180,E1 -6223.185,E2 -6223.185} C_VEL
LIN {X 0,Y 497.157,Z 542.638,A -85,B 0,C 180,E1 -6223.697,E2 -6223.697} C_VEL
LIN {X 0,Y 497.443,Z 529.794,A -85,B 0,C 180,E1 -6224.106,E2 -6224.106} C_VEL
LIN {X 0,Y 497.71,Z 514.921,A -85,B 0,C 180,E1 -6224.385,E2 -6224.385} C_VEL
LIN {X 0,Y 498.181,Z 432.08,A -85,B 0,C 180,E1 -6225.672,E2 -6225.672} C_VEL
LIN {X 0,Y 496.215,Z 413.492,A -85,B 0,C 180,E1 -6226.046,E2 -6226.046} C_VEL
LIN {X 0,Y 496.744,Z 390.268,A -85,B 0,C 180,E1 -6228.99,E2 -6228.99} C_VEL
LIN {X 0,Y 497.314,Z 365.303,A -85,B 0,C 180,E1 -6232.212,E2 -6232.212} C_VEL
LIN {X 0,Y 497.91,Z 345.469,A -85,B 0,C 180,E1 -6234.83,E2 -6234.83} C_VEL
LIN {X 0,Y 498.266,Z 332.373,A -85,B 0,C 180,E1 -6236.605,E2 -6236.605} C_VEL
LIN {X 0,Y 496.137,Z 321.457,A -85,B 0,C 180,E1 -6238.243,E2 -6238.243} C_VEL
LIN {X 0,Y 495.755,Z 319.735,A -85,B 0,C 180,E1 -6238.522,E2 -6238.522} C_VEL
LIN {X 0,Y 495.758,Z 319.733,A -85,B 0,C 180,E1 -6241.636,E2 -6241.636} C_VEL
LIN {X 0,Y 495.773,Z 319.732,A -85,B 0,C 180,E1 -6244.544,E2 -6244.544} C_VEL
LIN {X 0,Y 495.724,Z 319.734,A -85,B 0,C 180,E1 -6247.562,E2 -6247.562} C_VEL
LIN {X 0,Y 495.746,Z 319.736,A -85,B 0,C 180,E1 -6250.045,E2 -6250.045} C_VEL
LIN {X 0,Y 495.706,Z 319.736,A -85,B 0,C 180,E1 -6252.885,E2 -6252.885} C_VEL
LIN {X 0,Y 495.725,Z 319.738,A -85,B 0,C 180,E1 -6255.998,E2 -6255.998} C_VEL
LIN {X 0,Y 495.733,Z 319.732,A -85,B 0,C 180,E1 -6259.296,E2 -6259.296} C_VEL
LIN {X 0,Y 495.726,Z 319.733,A -85,B 0,C 180,E1 -6261.406,E2 -6261.406} C_VEL
LIN {X 0,Y 495.73,Z 319.733,A -85,B 0,C 180,E1 -6264.46,E2 -6264.46} C_VEL
LIN {X 0,Y 495.753,Z 319.73,A -85,B 0,C 180,E1 -6267.404,E2 -6267.404} C_VEL
LIN {X 0,Y 495.743,Z 319.733,A -85,B 0,C 180,E1 -6270.252,E2 -6270.252} C_VEL
LIN {X 0,Y 495.723,Z 319.735,A -85,B 0,C 180,E1 -6273.275,E2 -6273.275} C_VEL
LIN {X 0,Y 495.706,Z 319.742,A -85,B 0,C 180,E1 -6275.722,E2 -6275.722} C_VEL
LIN {X 0,Y 495.727,Z 319.734,A -85,B 0,C 180,E1 -6278.37,E2 -6278.37} C_VEL
LIN {X 0,Y 495.752,Z 319.732,A -85,B 0,C 180,E1 -6280.97,E2 -6280.97} C_VEL
LIN {X 0,Y 495.825,Z 319.724,A -85,B 0,C 180,E1 -6284.549,E2 -6284.549} C_VEL
LIN {X 0,Y 495.783,Z 319.767,A -85,B 0,C 180,E1 -6286.327,E2 -6286.327} C_VEL
LIN {X 0,Y 498.514,Z 328.28,A -85,B 0,C 180,E1 -6286.569,E2 -6286.569} C_VEL
LIN {X 0,Y 497.757,Z 410.623,A -85,B 0,C 180,E1 -6287.902,E2 -6287.902} C_VEL
LIN {X 0,Y 497.706,Z 423.76,A -85,B 0,C 180,E1 -6288.288,E2 -6288.288} C_VEL
LIN {X 0,Y 497.524,Z 435.776,A -85,B 0,C 180,E1 -6288.8,E2 -6288.8} C_VEL
LIN {X 0,Y 497.307,Z 446.603,A -85,B 0,C 180,E1 -6289.413,E2 -6289.413} C_VEL
LIN {X 0,Y 496.979,Z 457.917,A -85,B 0,C 180,E1 -6290.229,E2 -6290.229} C_VEL
LIN {X 0,Y 496.724,Z 468.1,A -85,B 0,C 180,E1 -6291.149,E2 -6291.149} C_VEL
LIN {X 0,Y 496.366,Z 476.984,A -85,B 0,C 180,E1 -6292.135,E2 -6292.135} C_VEL
LIN {X 0,Y 496.068,Z 485.526,A -85,B 0,C 180,E1 -6293.31,E2 -6293.31} C_VEL
LIN {X 0,Y 495.981,Z 492.546,A -85,B 0,C 180,E1 -6294.511,E2 -6294.511} C_VEL
LIN {X 0,Y 495.707,Z 497.411,A -85,B 0,C 180,E1 -6295.527,E2 -6295.527} C_VEL
LIN {X 0,Y 495.494,Z 502.102,A -85,B 0,C 180,E1 -6296.747,E2 -6296.747} C_VEL
LIN {X 0,Y 495.488,Z 505.657,A -85,B 0,C 180,E1 -6297.967,E2 -6297.967} C_VEL
LIN {X 0,Y 495.326,Z 508.224,A -85,B 0,C 180,E1 -6299.187,E2 -6299.187} C_VEL
LIN {X 0,Y 495.301,Z 509.409,A -85,B 0,C 180,E1 -6300,E2 -6300} C_VEL
LIN {X 0,Y 495.308,Z 510.185,A -85,B 0,C 180,E1 -6300.813,E2 -6300.813} C_VEL
LIN {X 0,Y 495.191,Z 510.545,A -85,B 0,C 180,E1 -6301.626,E2 -6301.626} C_VEL
LIN {X 0,Y 495.289,Z 510.073,A -85,B 0,C 180,E1 -6303.253,E2 -6303.253} C_VEL
LIN {X 0,Y 495.315,Z 509.241,A -85,B 0,C 180,E1 -6304.068,E2 -6304.068} C_VEL
LIN {X 0,Y 495.323,Z 507.981,A -85,B 0,C 180,E1 -6304.883,E2 -6304.883} C_VEL
LIN {X 0,Y 495.449,Z 505.314,A -85,B 0,C 180,E1 -6306.107,E2 -6306.107} C_VEL
LIN {X 0,Y 495.555,Z 501.63,A -85,B 0,C 180,E1 -6307.333,E2 -6307.333} C_VEL
LIN {X 0,Y 495.658,Z 496.817,A -85,B 0,C 180,E1 -6308.562,E2 -6308.562} C_VEL
LIN {X 0,Y 495.847,Z 490.718,A -85,B 0,C 180,E1 -6309.792,E2 -6309.792} C_VEL
LIN {X 0,Y 496.089,Z 483.114,A -85,B 0,C 180,E1 -6311.025,E2 -6311.025} C_VEL
LIN {X 0,Y 496.312,Z 474.87,A -85,B 0,C 180,E1 -6312.107,E2 -6312.107} C_VEL
LIN {X 0,Y 496.667,Z 464.654,A -85,B 0,C 180,E1 -6313.189,E2 -6313.189} C_VEL
LIN {X 0,Y 496.987,Z 453.761,A -85,B 0,C 180,E1 -6314.119,E2 -6314.119} C_VEL
LIN {X 0,Y 497.296,Z 443.075,A -85,B 0,C 180,E1 -6314.841,E2 -6314.841} C_VEL
LIN {X 0,Y 497.591,Z 430.196,A -85,B 0,C 180,E1 -6315.514,E2 -6315.514} C_VEL
LIN {X 0,Y 497.776,Z 417.349,A -85,B 0,C 180,E1 -6316.001,E2 -6316.001} C_VEL
LIN {X 0,Y 497.873,Z 404.945,A -85,B 0,C 180,E1 -6316.307,E2 -6316.307} C_VEL
LIN {X 0,Y 498.371,Z 327.645,A -85,B 0,C 180,E1 -6317.51,E2 -6317.51} C_VEL
LIN {X 0,Y 495.812,Z 319.724,A -85,B 0,C 180,E1 -6317.719,E2 -6317.719} C_VEL
LIN {X 0,Y 495.776,Z 319.733,A -85,B 0,C 180,E1 -6320.756,E2 -6320.756} C_VEL
LIN {X 0,Y 495.748,Z 319.729,A -85,B 0,C 180,E1 -6323.387,E2 -6323.387} C_VEL
LIN {X 0,Y 495.791,Z 319.725,A -85,B 0,C 180,E1 -6326.067,E2 -6326.067} C_VEL
LIN {X 0,Y 495.772,Z 319.731,A -85,B 0,C 180,E1 -6328.814,E2 -6328.814} C_VEL
LIN {X 0,Y 495.754,Z 319.728,A -85,B 0,C 180,E1 -6331.725,E2 -6331.725} C_VEL
LIN {X 0,Y 495.762,Z 319.733,A -85,B 0,C 180,E1 -6334.692,E2 -6334.692} C_VEL
LIN {X 0,Y 495.728,Z 319.731,A -85,B 0,C 180,E1 -6337.561,E2 -6337.561} C_VEL
LIN {X 0,Y 495.765,Z 319.732,A -85,B 0,C 180,E1 -6340.699,E2 -6340.699} C_VEL
LIN {X 0,Y 495.727,Z 319.734,A -85,B 0,C 180,E1 -6344.001,E2 -6344.001} C_VEL
LIN {X 0,Y 495.724,Z 319.733,A -85,B 0,C 180,E1 -6347.116,E2 -6347.116} C_VEL
LIN {X 0,Y 495.751,Z 319.73,A -85,B 0,C 180,E1 -6348.94,E2 -6348.94} C_VEL
LIN {X 0,Y 495.091,Z 319.811,A -85,B 0,C 180,E1 -6349.618,E2 -6349.618} C_VEL
LIN {X 0,Y 492.223,Z 320.172,A -85,B 0,C 180,E1 -6350.719,E2 -6350.719} C_VEL
LIN {X 0,Y 489.794,Z 320.476,A -85,B 0,C 180,E1 -6351.605,E2 -6351.605} C_VEL
LIN {X 0,Y 488.755,Z 320.605,A -85,B 0,C 180,E1 -6352.29,E2 -6352.29} C_VEL
LIN {X 0,Y 488.673,Z 320.613,A -85,B 0,C 180,E1 -6352.523,E2 -6352.523} C_VEL
LIN {X 0,Y 488.733,Z 320.605,A -85,B 0,C 180,E1 -6355.887,E2 -6355.887} C_VEL
LIN {X 0,Y 488.691,Z 320.61,A -85,B 0,C 180,E1 -6358.82,E2 -6358.82} C_VEL
LIN {X 0,Y 488.743,Z 320.603,A -85,B 0,C 180,E1 -6361.671,E2 -6361.671} C_VEL
LIN {X 0,Y 488.745,Z 320.607,A -85,B 0,C 180,E1 -6364.444,E2 -6364.444} C_VEL
LIN {X 0,Y 488.722,Z 320.604,A -85,B 0,C 180,E1 -6367.153,E2 -6367.153} C_VEL
LIN {X 0,Y 488.723,Z 320.607,A -85,B 0,C 180,E1 -6369.81,E2 -6369.81} C_VEL
LIN {X 0,Y 488.732,Z 320.608,A -85,B 0,C 180,E1 -6372.423,E2 -6372.423} C_VEL
LIN {X 0,Y 488.76,Z 320.6,A -85,B 0,C 180,E1 -6375,E2 -6375} C_VEL
LIN {X 0,Y 488.803,Z 320.599,A -85,B 0,C 180,E1 -6378.388,E2 -6378.388} C_VEL
LIN {X 0,Y 488.815,Z 320.596,A -85,B 0,C 180,E1 -6381.734,E2 -6381.734} C_VEL
LIN {X 0,Y 488.853,Z 320.594,A -85,B 0,C 180,E1 -6384.224,E2 -6384.224} C_VEL
LIN {X 0,Y 488.96,Z 320.577,A -85,B 0,C 180,E1 -6387.529,E2 -6387.529} C_VEL
LIN {X 0,Y 488.952,Z 320.576,A -85,B 0,C 180,E1 -6390.824,E2 -6390.824} C_VEL
LIN {X 0,Y 488.959,Z 320.577,A -85,B 0,C 180,E1 -6392.472,E2 -6392.472} C_VEL
LIN {X 0,Y 488.853,Z 320.592,A -85,B 0,C 180,E1 -6395.776,E2 -6395.776} C_VEL
LIN {X 0,Y 488.815,Z 320.597,A -85,B 0,C 180,E1 -6398.267,E2 -6398.267} C_VEL
LIN {X 0,Y 488.804,Z 320.597,A -85,B 0,C 180,E1 -6401.613,E2 -6401.613} C_VEL
LIN {X 0,Y 488.76,Z 320.6,A -85,B 0,C 180,E1 -6405.001,E2 -6405.001} C_VEL
LIN {X 0,Y 488.753,Z 320.602,A -85,B 0,C 180,E1 -6408.442,E2 -6408.442} C_VEL
LIN {X 0,Y 488.706,Z 320.607,A -85,B 0,C 180,E1 -6411.071,E2 -6411.071} C_VEL
LIN {X 0,Y 488.693,Z 320.613,A -85,B 0,C 180,E1 -6413.746,E2 -6413.746} C_VEL
LIN {X 0,Y 488.791,Z 320.596,A -85,B 0,C 180,E1 -6416.944,E2 -6416.944} C_VEL
LIN {X 0,Y 488.709,Z 320.607,A -85,B 0,C 180,E1 -6420.363,E2 -6420.363} C_VEL
LIN {X 0,Y 488.735,Z 320.607,A -85,B 0,C 180,E1 -6423.485,E2 -6423.485} C_VEL
LIN {X 0,Y 488.688,Z 320.61,A -85,B 0,C 180,E1 -6426.356,E2 -6426.356} C_VEL
LIN {X 0,Y 488.701,Z 320.61,A -85,B 0,C 180,E1 -6429.255,E2 -6429.255} C_VEL
LIN {X 0,Y 488.707,Z 320.612,A -85,B 0,C 180,E1 -6431.6,E2 -6431.6} C_VEL
LIN {X 0,Y 488.701,Z 320.607,A -85,B 0,C 180,E1 -6434.803,E2 -6434.803} C_VEL
LIN {X 0,Y 488.692,Z 320.613,A -85,B 0,C 180,E1 -6437.475,E2 -6437.475} C_VEL
LIN {X 0,Y 488.734,Z 320.61,A -85,B 0,C 180,E1 -6439.677,E2 -6439.677} C_VEL
LIN {X 0,Y 488.68,Z 320.611,A -85,B 0,C 180,E1 -6442.842,E2 -6442.842} C_VEL
LIN {X 0,Y 488.725,Z 320.607,A -85,B 0,C 180,E1 -6445.887,E2 -6445.887} C_VEL
LIN {X 0,Y 488.693,Z 320.609,A -85,B 0,C 180,E1 -6448.821,E2 -6448.821} C_VEL
LIN {X 0,Y 488.746,Z 320.607,A -85,B 0,C 180,E1 -6451.672,E2 -6451.672} C_VEL
LIN {X 0,Y 488.742,Z 320.601,A -85,B 0,C 180,E1 -6454.444,E2 -6454.444} C_VEL
LIN {X 0,Y 488.754,Z 320.696,A -85,B 0,C 180,E1 -6456.158,E2 -6456.158} C_VEL
LIN {X 0,Y 491.607,Z 329.997,A -85,B 0,C 180,E1 -6456.404,E2 -6456.404} C_VEL
LIN {X 0,Y 490.96,Z 408.648,A -85,B 0,C 180,E1 -6457.652,E2 -6457.652} C_VEL
LIN {X 0,Y 490.789,Z 420.375,A -85,B 0,C 180,E1 -6457.976,E2 -6457.976} C_VEL
LIN {X 0,Y 490.666,Z 432.171,A -85,B 0,C 180,E1 -6458.45,E2 -6458.45} C_VEL
LIN {X 0,Y 490.382,Z 444.401,A -85,B 0,C 180,E1 -6459.115,E2 -6459.115} C_VEL
LIN {X 0,Y 490.068,Z 455.23,A -85,B 0,C 180,E1 -6459.869,E2 -6459.869} C_VEL
LIN {X 0,Y 489.757,Z 465.184,A -85,B 0,C 180,E1 -6460.729,E2 -6460.729} C_VEL
LIN {X 0,Y 489.414,Z 475.179,A -85,B 0,C 180,E1 -6461.801,E2 -6461.801} C_VEL
LIN {X 0,Y 489.113,Z 483.325,A -85,B 0,C 180,E1 -6462.869,E2 -6462.869} C_VEL
LIN {X 0,Y 488.835,Z 491.238,A -85,B 0,C 180,E1 -6464.148,E2 -6464.148} C_VEL
LIN {X 0,Y 488.627,Z 497.484,A -85,B 0,C 180,E1 -6465.422,E2 -6465.422} C_VEL
LIN {X 0,Y 488.45,Z 502.396,A -85,B 0,C 180,E1 -6466.691,E2 -6466.691} C_VEL
LIN {X 0,Y 488.395,Z 506.508,A -85,B 0,C 180,E1 -6468.105,E2 -6468.105} C_VEL
LIN {X 0,Y 488.289,Z 508.809,A -85,B 0,C 180,E1 -6469.216,E2 -6469.216} C_VEL
LIN {X 0,Y 488.225,Z 510.07,A -85,B 0,C 180,E1 -6470.053,E2 -6470.053} C_VEL
LIN {X 0,Y 488.246,Z 510.873,A -85,B 0,C 180,E1 -6470.89,E2 -6470.89} C_VEL
LIN {X 0,Y 488.279,Z 511.275,A -85,B 0,C 180,E1 -6472.557,E2 -6472.557} C_VEL
LIN {X 0,Y 488.314,Z 510.867,A -85,B 0,C 180,E1 -6473.389,E2 -6473.389} C_VEL
LIN {X 0,Y 488.391,Z 508.807,A -85,B 0,C 180,E1 -6475.047,E2 -6475.047} C_VEL
LIN {X 0,Y 488.425,Z 506.174,A -85,B 0,C 180,E1 -6476.288,E2 -6476.288} C_VEL
LIN {X 0,Y 488.539,Z 502.52,A -85,B 0,C 180,E1 -6477.527,E2 -6477.527} C_VEL
LIN {X 0,Y 488.695,Z 497.752,A -85,B 0,C 180,E1 -6478.764,E2 -6478.764} C_VEL
LIN {X 0,Y 488.937,Z 491.706,A -85,B 0,C 180,E1 -6480,E2 -6480} C_VEL
LIN {X 0,Y 489.205,Z 484.13,A -85,B 0,C 180,E1 -6481.235,E2 -6481.235} C_VEL
LIN {X 0,Y 489.567,Z 474.706,A -85,B 0,C 180,E1 -6482.469,E2 -6482.469} C_VEL
LIN {X 0,Y 489.914,Z 464.825,A -85,B 0,C 180,E1 -6483.496,E2 -6483.496} C_VEL
LIN {X 0,Y 490.13,Z 455.146,A -85,B 0,C 180,E1 -6484.318,E2 -6484.318} C_VEL
LIN {X 0,Y 490.471,Z 444.62,A -85,B 0,C 180,E1 -6485.035,E2 -6485.035} C_VEL
LIN {X 0,Y 490.715,Z 433.063,A -85,B 0,C 180,E1 -6485.651,E2 -6485.651} C_VEL
LIN {X 0,Y 490.85,Z 419.824,A -85,B 0,C 180,E1 -6486.165,E2 -6486.165} C_VEL
LIN {X 0,Y 490.957,Z 407.831,A -85,B 0,C 180,E1 -6486.473,E2 -6486.473} C_VEL
LIN {X 0,Y 491.675,Z 329.112,A -85,B 0,C 180,E1 -6487.743,E2 -6487.743} C_VEL
LIN {X 0,Y 488.791,Z 320.601,A -85,B 0,C 180,E1 -6488.013,E2 -6488.013} C_VEL
LIN {X 0,Y 488.777,Z 320.6,A -85,B 0,C 180,E1 -6491.614,E2 -6491.614} C_VEL
LIN {X 0,Y 488.758,Z 320.604,A -85,B 0,C 180,E1 -6495.001,E2 -6495.001} C_VEL
LIN {X 0,Y 488.707,Z 320.613,A -85,B 0,C 180,E1 -6498.444,E2 -6498.444} C_VEL
LIN {X 0,Y 488.681,Z 320.612,A -85,B 0,C 180,E1 -6501.072,E2 -6501.072} C_VEL
LIN {X 0,Y 488.667,Z 320.613,A -85,B 0,C 180,E1 -6503.747,E2 -6503.747} C_VEL
LIN {X 0,Y 488.672,Z 320.617,A -85,B 0,C 180,E1 -6506.477,E2 -6506.477} C_VEL
LIN {X 0,Y 488.694,Z 320.608,A -85,B 0,C 180,E1 -6509.273,E2 -6509.273} C_VEL
LIN {X 0,Y 488.699,Z 320.613,A -85,B 0,C 180,E1 -6512.148,E2 -6512.148} C_VEL
LIN {X 0,Y 488.71,Z 320.604,A -85,B 0,C 180,E1 -6515.116,E2 -6515.116} C_VEL
LIN {X 0,Y 488.66,Z 320.616,A -85,B 0,C 180,E1 -6518.202,E2 -6518.202} C_VEL
LIN {X 0,Y 488.697,Z 320.608,A -85,B 0,C 180,E1 -6520.341,E2 -6520.341} C_VEL
LIN {X 0,Y 488.677,Z 320.614,A -85,B 0,C 180,E1 -6523.656,E2 -6523.656} C_VEL
LIN {X 0,Y 488.679,Z 320.612,A -85,B 0,C 180,E1 -6526.344,E2 -6526.344} C_VEL
LIN {X 0,Y 488.707,Z 320.613,A -85,B 0,C 180,E1 -6529.673,E2 -6529.673} C_VEL
LIN {X 0,Y 488.671,Z 320.611,A -85,B 0,C 180,E1 -6532.84,E2 -6532.84} C_VEL
LIN {X 0,Y 488.727,Z 320.609,A -85,B 0,C 180,E1 -6535.886,E2 -6535.886} C_VEL
LIN {X 0,Y 488.696,Z 320.609,A -85,B 0,C 180,E1 -6538.82,E2 -6538.82} C_VEL
LIN {X 0,Y 488.773,Z 320.731,A -85,B 0,C 180,E1 -6540.881,E2 -6540.881} C_VEL
LIN {X 0,Y 491.882,Z 334.988,A -85,B 0,C 180,E1 -6543.022,E2 -6543.022} C_VEL
LIN {X 0,Y 491.635,Z 346.564,A -85,B 0,C 180,E1 -6544.605,E2 -6544.605} C_VEL
